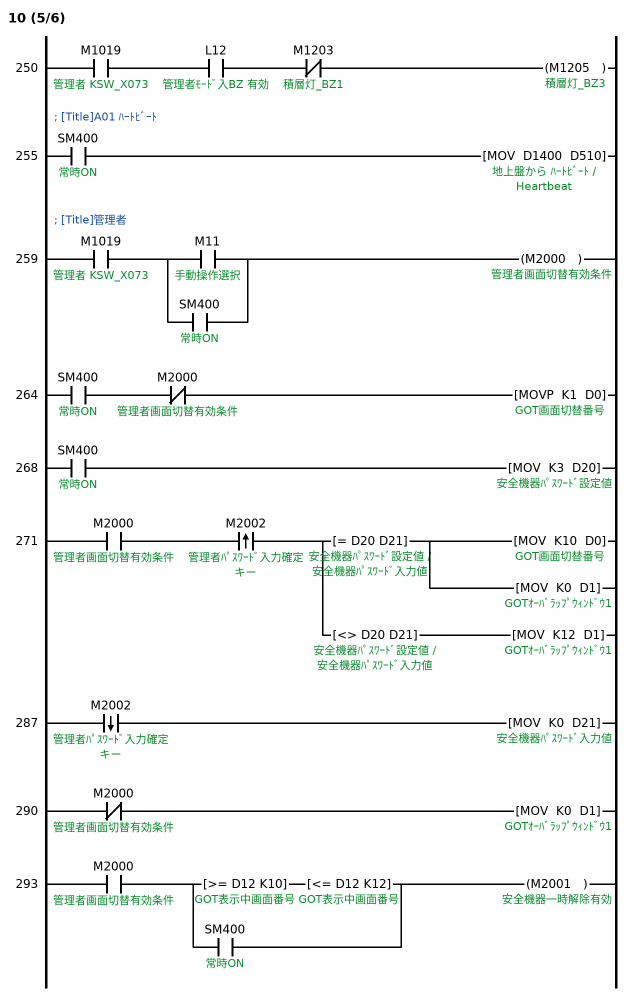
250   LD      M1019  ; 管理者 KSW_X073
      AND     L12  ; 管理者ﾓｰﾄﾞ入BZ 有効
      ANI     M1203  ; 積層灯_BZ1
      OUT     M1205  ; 積層灯_BZ3
; [Title]A01 ﾊｰﾄﾋﾞｰﾄ
255   LD      SM400  ; 常時ON
      MOV     D1400 D510  ; 地上盤から ﾊｰﾄﾋﾞｰﾄ / Heartbeat
; [Title]管理者
259   LD      M1019  ; 管理者 KSW_X073
      LD      M11  ; 手動操作選択
      OR      SM400  ; 常時ON
      ANB
      OUT     M2000  ; 管理者画面切替有効条件
264   LD      SM400  ; 常時ON
      ANI     M2000  ; 管理者画面切替有効条件
      MOVP    K1 D0  ; GOT画面切替番号
268   LD      SM400  ; 常時ON
      MOV     K3 D20  ; 安全機器ﾊﾟｽﾜｰﾄﾞ設定値
271   LD      M2000  ; 管理者画面切替有効条件
      ANDP    M2002  ; 管理者ﾊﾟｽﾜｰﾄﾞ入力確定キー
      MPS
      AND=    D20 D21  ; 安全機器ﾊﾟｽﾜｰﾄﾞ設定値 / 安全機器ﾊﾟｽﾜｰﾄﾞ入力値
      MOV     K10 D0
      MOV     K0 D1  ; GOTｵｰﾊﾞﾗｯﾌﾟｳｨﾝﾄﾞｳ1
      MPP
      AND<>   D20 D21  ; 安全機器ﾊﾟｽﾜｰﾄﾞ設定値 / 安全機器ﾊﾟｽﾜｰﾄﾞ入力値
      MOV     K12 D1
287   LDF     M2002  ; 管理者ﾊﾟｽﾜｰﾄﾞ入力確定キー
      MOV     K0 D21
290   LDI     M2000  ; 管理者画面切替有効条件
      MOV     K0 D1
293   LD      M2000  ; 管理者画面切替有効条件
      LD>=    D12 K10  ; GOT表示中画面番号
      AND<=   D12 K12  ; GOT表示中画面番号
      OR      SM400  ; 常時ON
      ANB
      OUT     M2001  ; 安全機器一時解除有効
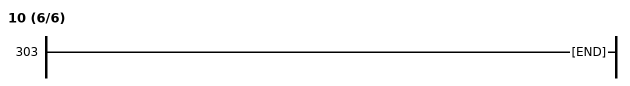
303   END
END_PROGRAM

PROGRAM 11  // 自動搬入
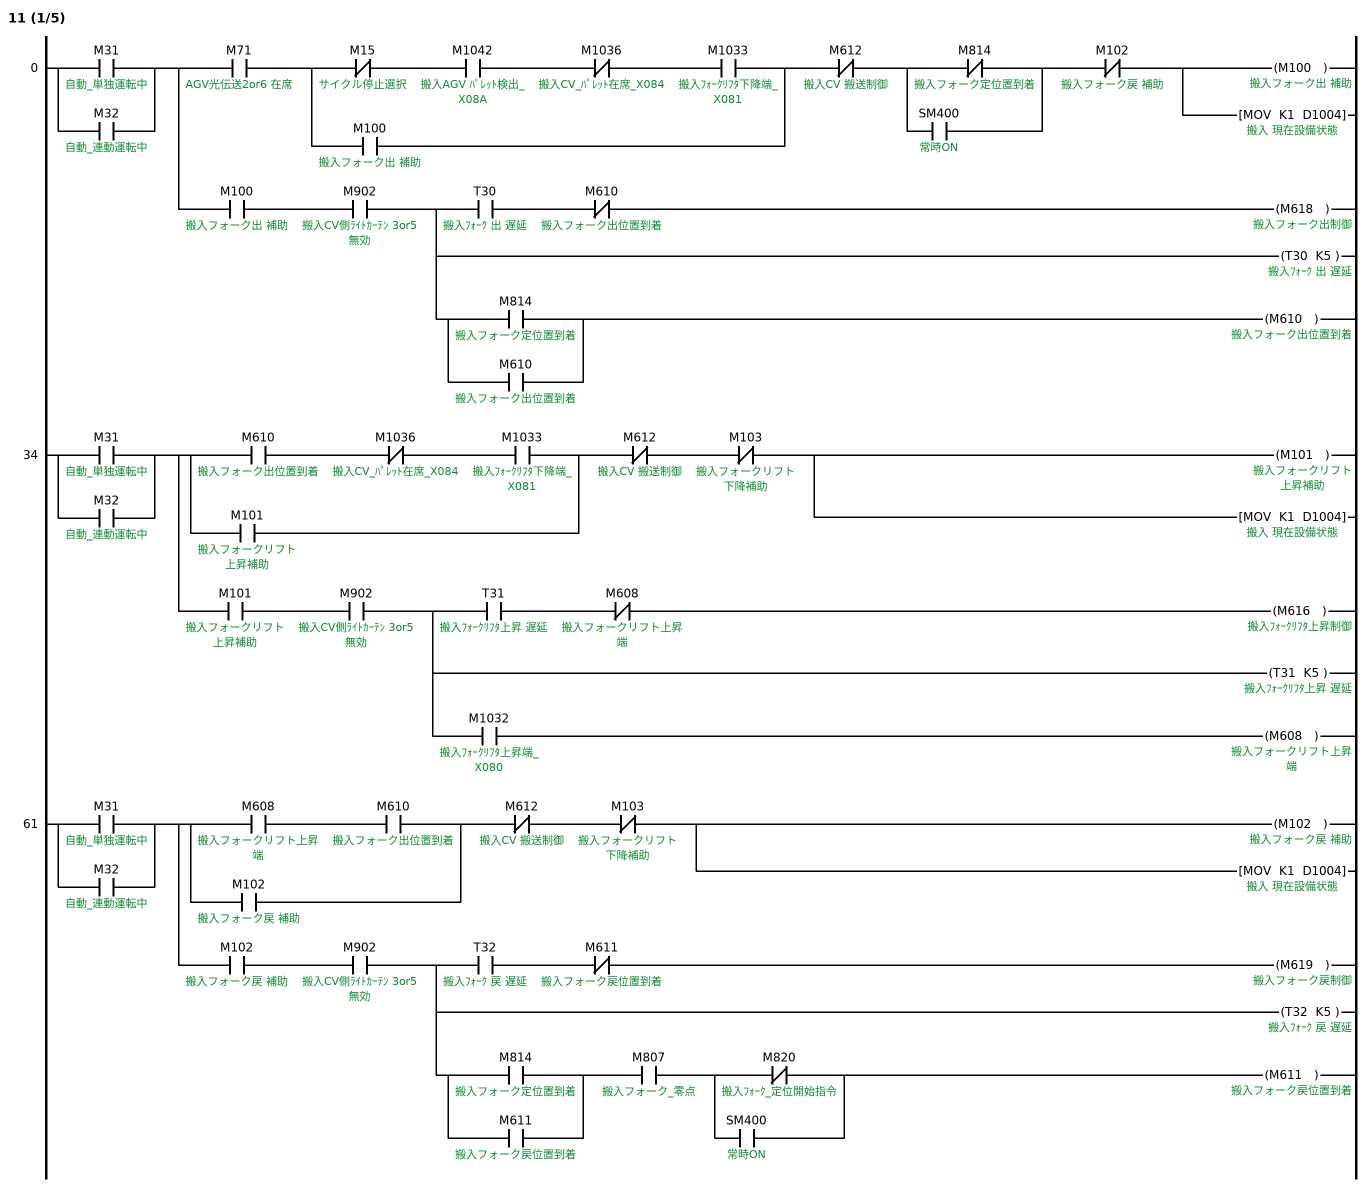
0     LD      M31  ; 自動_単独運転中
      OR      M32  ; 自動_連動運転中
      MPS
      AND     M71  ; AGV光伝送2or6 在席
      LDI     M15  ; サイクル停止選択
      AND     M1042  ; 搬入AGV ﾊﾟﾚｯﾄ検出_X08A
      ANI     M1036  ; 搬入CV_ﾊﾟﾚｯﾄ在席_X084
      AND     M1033  ; 搬入ﾌｫｰｸﾘﾌﾀ下降端_X081
      OR      M100  ; 搬入フォーク出 補助
      ANB
      ANI     M612  ; 搬入CV 搬送制御
      LDI     M814  ; 搬入フォーク定位置到着
      OR      SM400  ; 常時ON
      ANB
      ANI     M102  ; 搬入フォーク戻 補助
      OUT     M100  ; 搬入フォーク出 補助
      MOV     K1 D1004  ; 搬入 現在設備状態
      MPP
      AND     M100  ; 搬入フォーク出 補助
      AND     M902  ; 搬入CV側ﾗｲﾄｶｰﾃﾝ 3or5 無効
      MPS
      AND     T30  ; 搬入ﾌｫｰｸ 出 遅延
      ANI     M610  ; 搬入フォーク出位置到着
      OUT     M618  ; 搬入フォーク出制御
      MPP
      OUT     T30 K5  ; 搬入ﾌｫｰｸ 出 遅延
      LD      M814  ; 搬入フォーク定位置到着
      OR      M610  ; 搬入フォーク出位置到着
      ANB
      OUT     M610  ; 搬入フォーク出位置到着
34    LD      M31  ; 自動_単独運転中
      OR      M32  ; 自動_連動運転中
      MPS
      LD      M610  ; 搬入フォーク出位置到着
      ANI     M1036  ; 搬入CV_ﾊﾟﾚｯﾄ在席_X084
      AND     M1033  ; 搬入ﾌｫｰｸﾘﾌﾀ下降端_X081
      OR      M101  ; 搬入フォークリフト 上昇補助
      ANB
      ANI     M612  ; 搬入CV 搬送制御
      ANI     M103  ; 搬入フォークリフト 下降補助
      OUT     M101  ; 搬入フォークリフト 上昇補助
      MOV     K1 D1004
      MPP
      AND     M101  ; 搬入フォークリフト 上昇補助
      AND     M902  ; 搬入CV側ﾗｲﾄｶｰﾃﾝ 3or5 無効
      MPS
      AND     T31  ; 搬入ﾌｫｰｸﾘﾌﾀ上昇 遅延
      ANI     M608  ; 搬入フォークリフト上昇端
      OUT     M616  ; 搬入ﾌｫｰｸﾘﾌﾀ上昇制御
      MPP
      OUT     T31 K5  ; 搬入ﾌｫｰｸﾘﾌﾀ上昇 遅延
      AND     M1032  ; 搬入ﾌｫｰｸﾘﾌﾀ上昇端_X080
      OUT     M608  ; 搬入フォークリフト上昇端
61    LD      M31  ; 自動_単独運転中
      OR      M32  ; 自動_連動運転中
      MPS
      LD      M608  ; 搬入フォークリフト上昇端
      AND     M610  ; 搬入フォーク出位置到着
      OR      M102  ; 搬入フォーク戻 補助
      ANB
      ANI     M612  ; 搬入CV 搬送制御
      ANI     M103  ; 搬入フォークリフト 下降補助
      OUT     M102  ; 搬入フォーク戻 補助
      MOV     K1 D1004
      MPP
      AND     M102  ; 搬入フォーク戻 補助
      AND     M902  ; 搬入CV側ﾗｲﾄｶｰﾃﾝ 3or5 無効
      MPS
      AND     T32  ; 搬入ﾌｫｰｸ 戻 遅延
      ANI     M611  ; 搬入フォーク戻位置到着
      OUT     M619  ; 搬入フォーク戻制御
      MPP
      OUT     T32 K5  ; 搬入ﾌｫｰｸ 戻 遅延
      LD      M814  ; 搬入フォーク定位置到着
      OR      M611  ; 搬入フォーク戻位置到着
      ANB
      AND     M807  ; 搬入フォーク_零点
      LDI     M820  ; 搬入ﾌｫｰｸ_定位開始指令
      OR      SM400  ; 常時ON
      ANB
      OUT     M611  ; 搬入フォーク戻位置到着
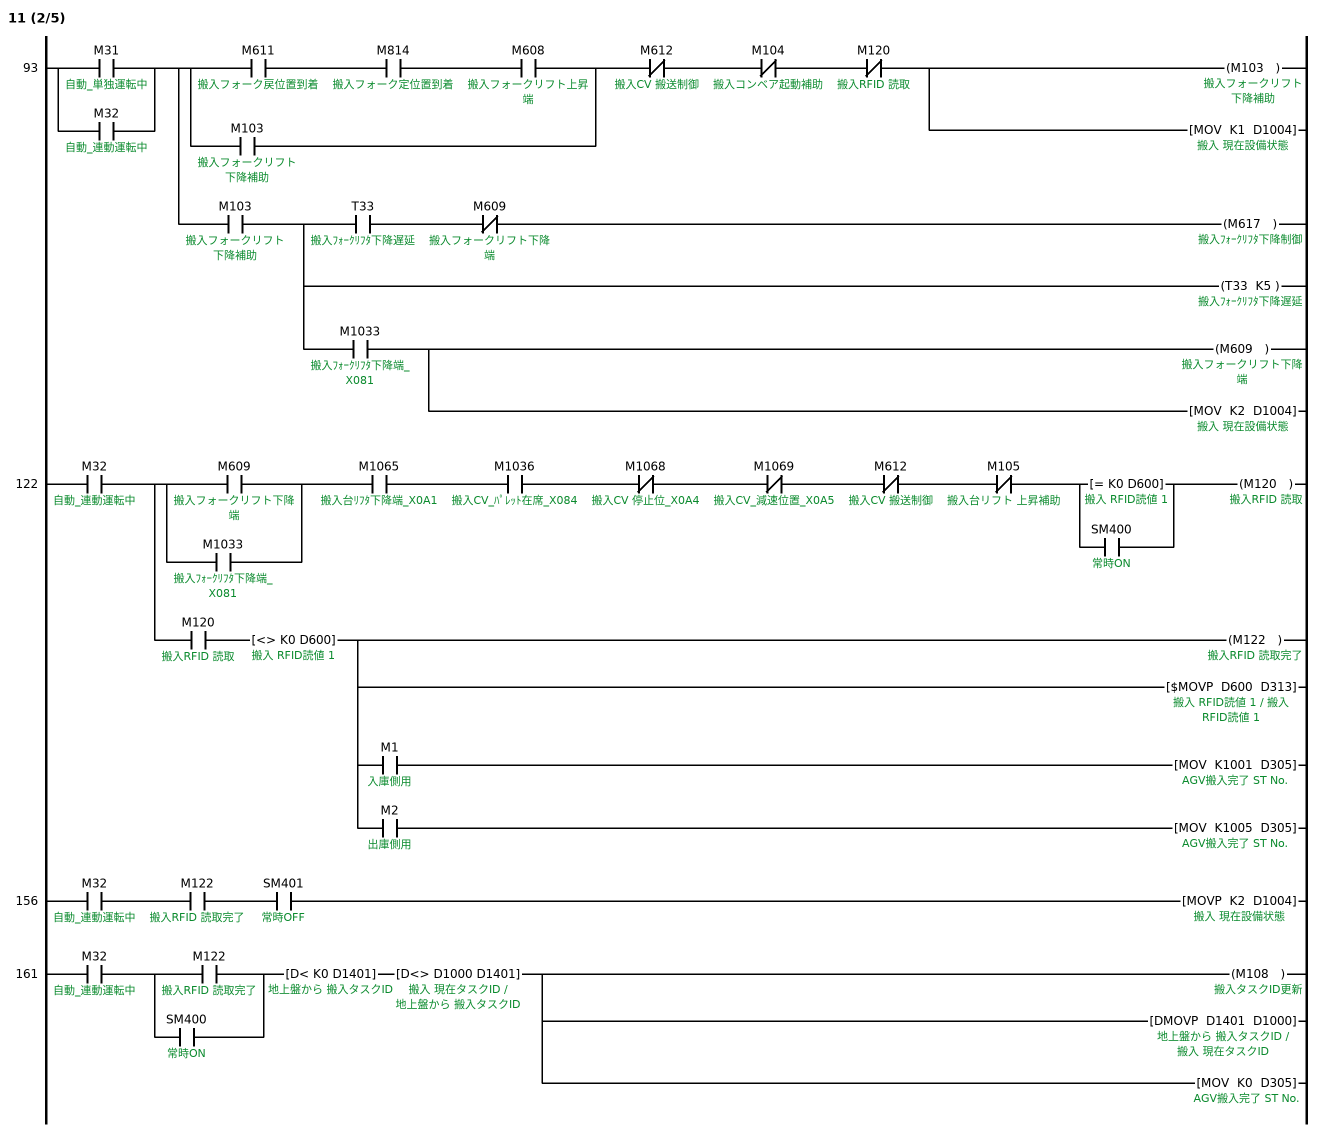
93    LD      M31  ; 自動_単独運転中
      OR      M32  ; 自動_連動運転中
      MPS
      LD      M611  ; 搬入フォーク戻位置到着
      AND     M814  ; 搬入フォーク定位置到着
      AND     M608  ; 搬入フォークリフト上昇端
      OR      M103  ; 搬入フォークリフト 下降補助
      ANB
      ANI     M612  ; 搬入CV 搬送制御
      ANI     M104  ; 搬入コンベア起動補助
      ANI     M120  ; 搬入RFID 読取
      OUT     M103  ; 搬入フォークリフト 下降補助
      MOV     K1 D1004
      MPP
      AND     M103  ; 搬入フォークリフト 下降補助
      MPS
      AND     T33  ; 搬入ﾌｫｰｸﾘﾌﾀ下降遅延
      ANI     M609  ; 搬入フォークリフト下降端
      OUT     M617  ; 搬入ﾌｫｰｸﾘﾌﾀ下降制御
      MPP
      OUT     T33 K5  ; 搬入ﾌｫｰｸﾘﾌﾀ下降遅延
      AND     M1033  ; 搬入ﾌｫｰｸﾘﾌﾀ下降端_X081
      OUT     M609  ; 搬入フォークリフト下降端
      MOV     K2 D1004
122   LD      M32  ; 自動_連動運転中
      MPS
      LD      M609  ; 搬入フォークリフト下降端
      OR      M1033  ; 搬入ﾌｫｰｸﾘﾌﾀ下降端_X081
      ANB
      AND     M1065  ; 搬入台ﾘﾌﾀ下降端_X0A1
      AND     M1036  ; 搬入CV_ﾊﾟﾚｯﾄ在席_X084
      ANI     M1068  ; 搬入CV 停止位_X0A4
      ANI     M1069  ; 搬入CV_減速位置_X0A5
      ANI     M612  ; 搬入CV 搬送制御
      ANI     M105  ; 搬入台リフト 上昇補助
      LD=     K0 D600  ; 搬入 RFID読値 1
      OR      SM400  ; 常時ON
      ANB
      OUT     M120  ; 搬入RFID 読取
      MPP
      AND     M120  ; 搬入RFID 読取
      AND<>   K0 D600  ; 搬入 RFID読値 1
      OUT     M122  ; 搬入RFID 読取完了
      $MOVP   D600 D313  ; 搬入 RFID読値 1
      MPS
      AND     M1  ; 入庫側用
      MOV     K1001 D305  ; AGV搬入完了 ST No.
      MPP
      AND     M2  ; 出庫側用
      MOV     K1005 D305
156   LD      M32  ; 自動_連動運転中
      AND     M122  ; 搬入RFID 読取完了
      AND     SM401  ; 常時OFF
      MOVP    K2 D1004
161   LD      M32  ; 自動_連動運転中
      LD      M122  ; 搬入RFID 読取完了
      OR      SM400  ; 常時ON
      ANB
      ANDD<   K0 D1401  ; 地上盤から 搬入タスクID
      ANDD<>  D1000 D1401  ; 搬入 現在タスクID / 地上盤から 搬入タスクID
      OUT     M108  ; 搬入タスクID更新
      DMOVP   D1401 D1000
      MOV     K0 D305
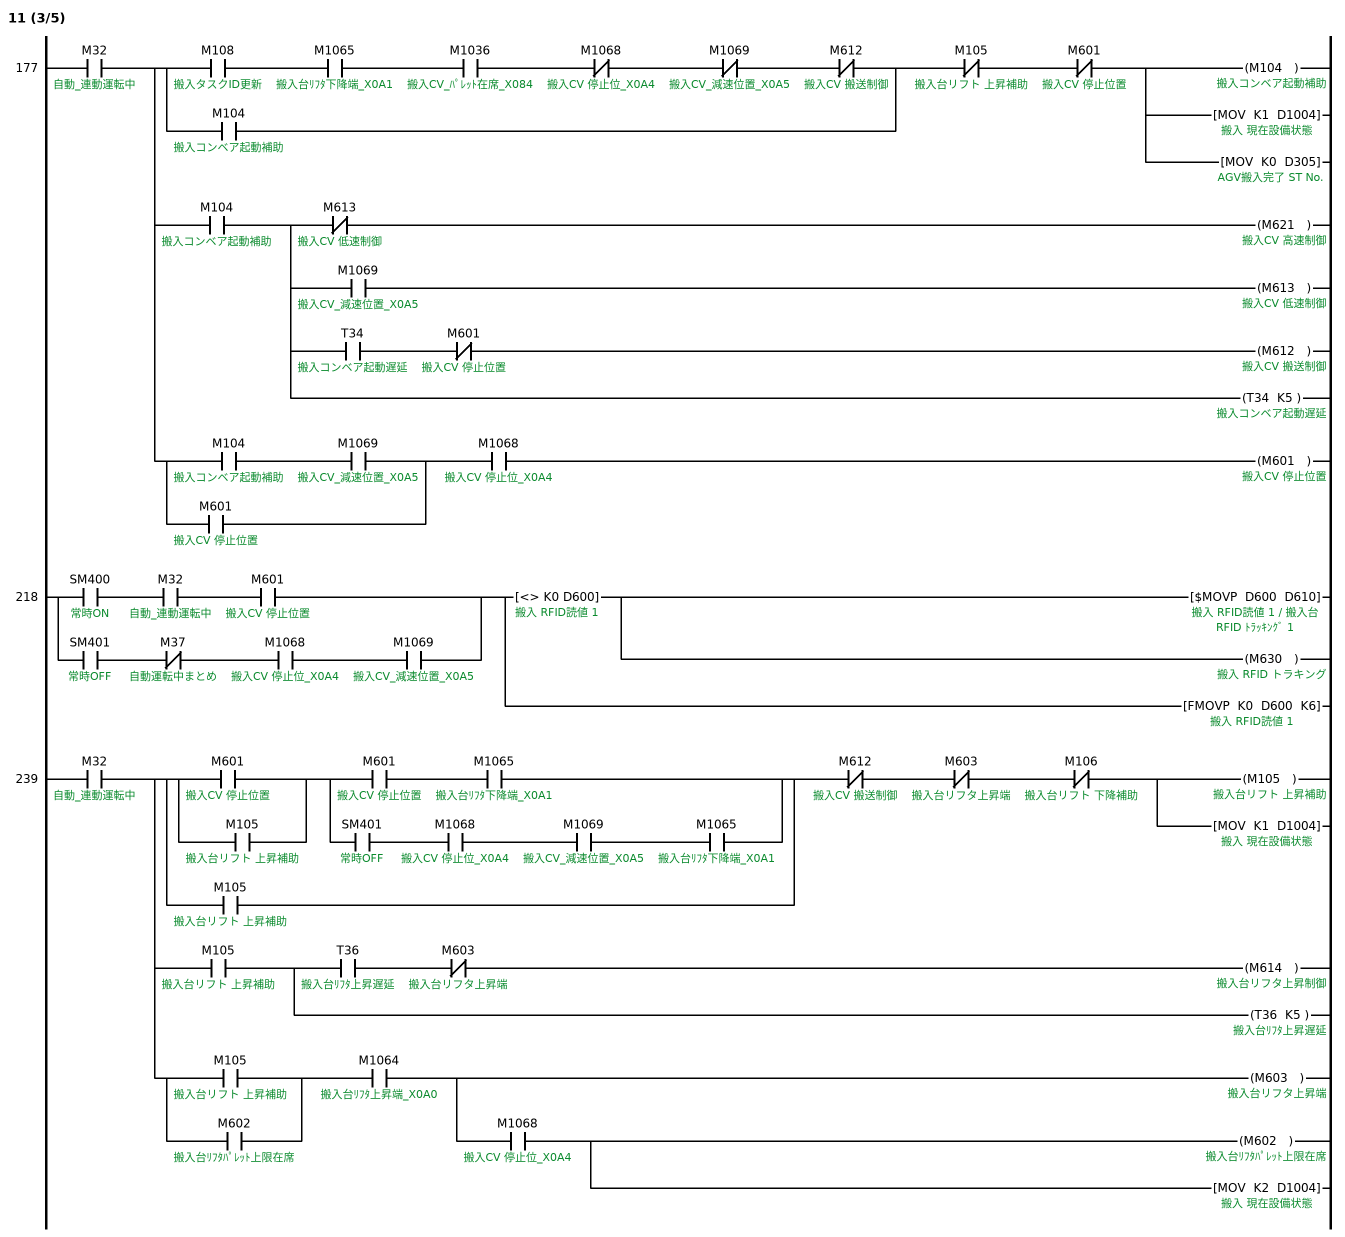
177   LD      M32  ; 自動_連動運転中
      MPS
      LD      M108  ; 搬入タスクID更新
      AND     M1065  ; 搬入台ﾘﾌﾀ下降端_X0A1
      AND     M1036  ; 搬入CV_ﾊﾟﾚｯﾄ在席_X084
      ANI     M1068  ; 搬入CV 停止位_X0A4
      ANI     M1069  ; 搬入CV_減速位置_X0A5
      ANI     M612  ; 搬入CV 搬送制御
      OR      M104  ; 搬入コンベア起動補助
      ANB
      ANI     M105  ; 搬入台リフト 上昇補助
      ANI     M601  ; 搬入CV 停止位置
      OUT     M104  ; 搬入コンベア起動補助
      MOV     K1 D1004
      MOV     K0 D305
      MRD
      AND     M104  ; 搬入コンベア起動補助
      MPS
      ANI     M613  ; 搬入CV 低速制御
      OUT     M621  ; 搬入CV 高速制御
      MRD
      AND     M1069  ; 搬入CV_減速位置_X0A5
      OUT     M613  ; 搬入CV 低速制御
      MRD
      AND     T34  ; 搬入コンベア起動遅延
      ANI     M601  ; 搬入CV 停止位置
      OUT     M612  ; 搬入CV 搬送制御
      MPP
      OUT     T34 K5  ; 搬入コンベア起動遅延
      MPP
      LD      M104  ; 搬入コンベア起動補助
      AND     M1069  ; 搬入CV_減速位置_X0A5
      OR      M601  ; 搬入CV 停止位置
      ANB
      AND     M1068  ; 搬入CV 停止位_X0A4
      OUT     M601  ; 搬入CV 停止位置
218   LD      SM400  ; 常時ON
      AND     M32  ; 自動_連動運転中
      AND     M601  ; 搬入CV 停止位置
      LD      SM401  ; 常時OFF
      ANI     M37  ; 自動運転中まとめ
      AND     M1068  ; 搬入CV 停止位_X0A4
      AND     M1069  ; 搬入CV_減速位置_X0A5
      ORB
      MPS
      AND<>   K0 D600  ; 搬入 RFID読値 1
      $MOVP   D600 D610  ; 搬入台 RFID ﾄﾗｯｷﾝｸﾞ 1
      OUT     M630  ; 搬入 RFID トラキング
      MPP
      FMOVP   K0 D600 K6
239   LD      M32  ; 自動_連動運転中
      MPS
      LD      M601  ; 搬入CV 停止位置
      OR      M105  ; 搬入台リフト 上昇補助
      LD      M601  ; 搬入CV 停止位置
      AND     M1065  ; 搬入台ﾘﾌﾀ下降端_X0A1
      LD      SM401  ; 常時OFF
      AND     M1068  ; 搬入CV 停止位_X0A4
      AND     M1069  ; 搬入CV_減速位置_X0A5
      AND     M1065  ; 搬入台ﾘﾌﾀ下降端_X0A1
      ORB
      ANB
      OR      M105  ; 搬入台リフト 上昇補助
      ANB
      ANI     M612  ; 搬入CV 搬送制御
      ANI     M603  ; 搬入台リフタ上昇端
      ANI     M106  ; 搬入台リフト 下降補助
      OUT     M105  ; 搬入台リフト 上昇補助
      MOV     K1 D1004
      MRD
      AND     M105  ; 搬入台リフト 上昇補助
      MPS
      AND     T36  ; 搬入台ﾘﾌﾀ上昇遅延
      ANI     M603  ; 搬入台リフタ上昇端
      OUT     M614  ; 搬入台リフタ上昇制御
      MPP
      OUT     T36 K5  ; 搬入台ﾘﾌﾀ上昇遅延
      MPP
      LD      M105  ; 搬入台リフト 上昇補助
      OR      M602  ; 搬入台ﾘﾌﾀﾊﾟﾚｯﾄ上限在席
      ANB
      AND     M1064  ; 搬入台ﾘﾌﾀ上昇端_X0A0
      OUT     M603  ; 搬入台リフタ上昇端
      AND     M1068  ; 搬入CV 停止位_X0A4
      OUT     M602  ; 搬入台ﾘﾌﾀﾊﾟﾚｯﾄ上限在席
      MOV     K2 D1004
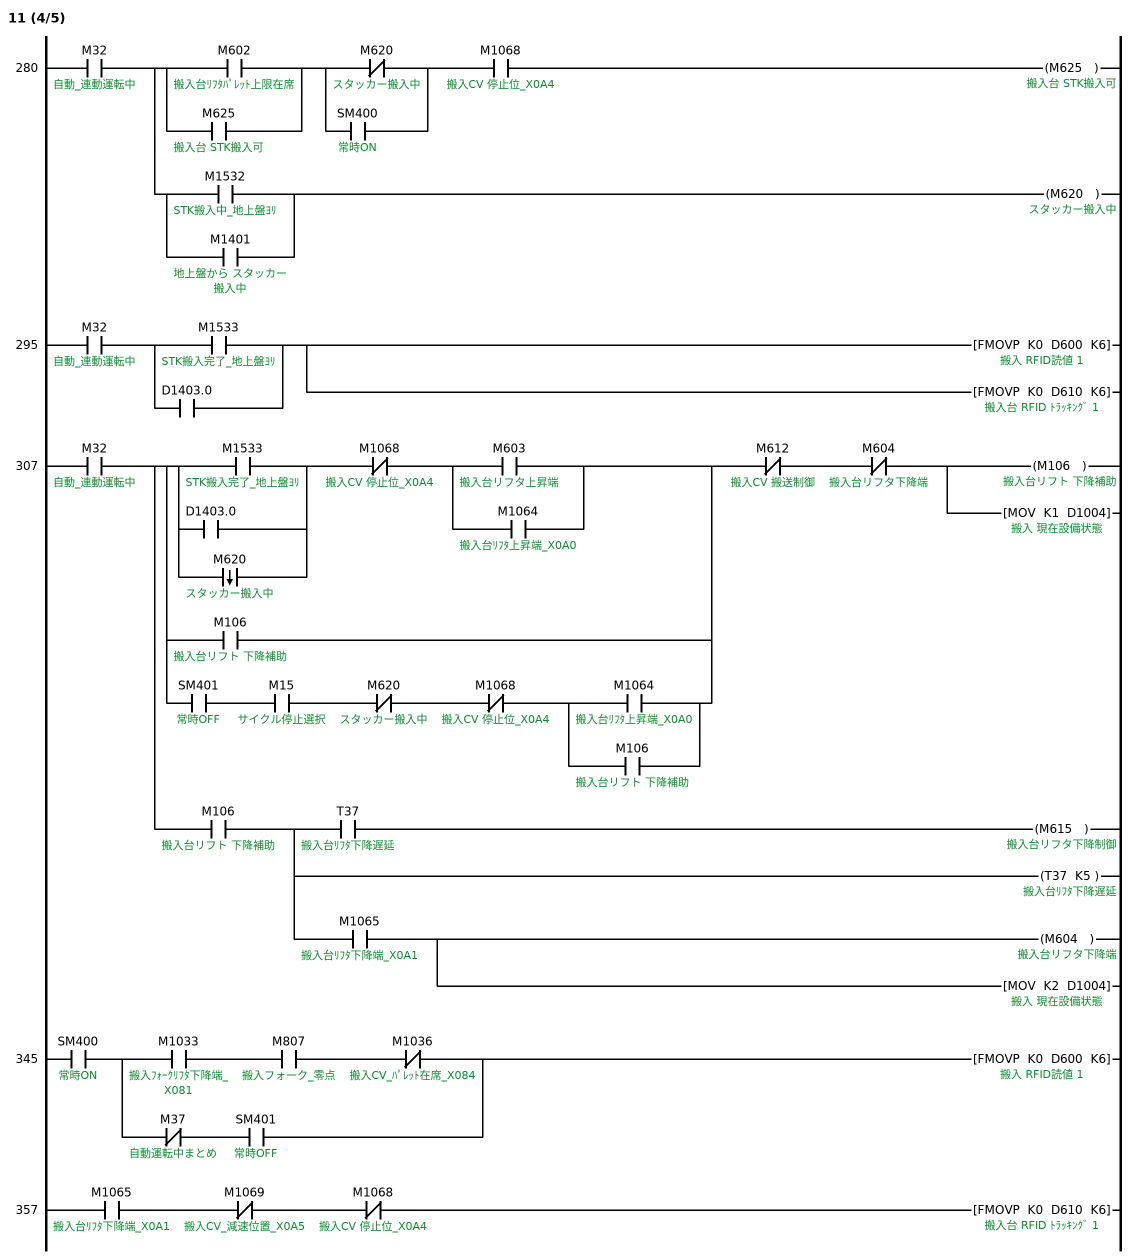
280   LD      M32  ; 自動_連動運転中
      MPS
      LD      M602  ; 搬入台ﾘﾌﾀﾊﾟﾚｯﾄ上限在席
      OR      M625  ; 搬入台 STK搬入可
      ANB
      LDI     M620  ; スタッカー搬入中
      OR      SM400  ; 常時ON
      ANB
      AND     M1068  ; 搬入CV 停止位_X0A4
      OUT     M625  ; 搬入台 STK搬入可
      MPP
      LD      M1532  ; STK搬入中_地上盤ﾖﾘ
      OR      M1401  ; 地上盤から スタッカー 搬入中
      ANB
      OUT     M620  ; スタッカー搬入中
295   LD      M32  ; 自動_連動運転中
      LD      M1533  ; STK搬入完了_地上盤ﾖﾘ
      OR      D1403.0
      ANB
      FMOVP   K0 D600 K6
      FMOVP   K0 D610 K6
307   LD      M32  ; 自動_連動運転中
      MPS
      LD      M1533  ; STK搬入完了_地上盤ﾖﾘ
      OR      D1403.0
      ORF     M620  ; スタッカー搬入中
      ANI     M1068  ; 搬入CV 停止位_X0A4
      LD      M603  ; 搬入台リフタ上昇端
      OR      M1064  ; 搬入台ﾘﾌﾀ上昇端_X0A0
      ANB
      OR      M106  ; 搬入台リフト 下降補助
      LD      SM401  ; 常時OFF
      AND     M15  ; サイクル停止選択
      ANI     M620  ; スタッカー搬入中
      ANI     M1068  ; 搬入CV 停止位_X0A4
      LD      M1064  ; 搬入台ﾘﾌﾀ上昇端_X0A0
      OR      M106  ; 搬入台リフト 下降補助
      ANB
      ORB
      ANB
      ANI     M612  ; 搬入CV 搬送制御
      ANI     M604  ; 搬入台リフタ下降端
      OUT     M106  ; 搬入台リフト 下降補助
      MOV     K1 D1004
      MPP
      AND     M106  ; 搬入台リフト 下降補助
      MPS
      AND     T37  ; 搬入台ﾘﾌﾀ下降遅延
      OUT     M615  ; 搬入台リフタ下降制御
      MPP
      OUT     T37 K5  ; 搬入台ﾘﾌﾀ下降遅延
      AND     M1065  ; 搬入台ﾘﾌﾀ下降端_X0A1
      OUT     M604  ; 搬入台リフタ下降端
      MOV     K2 D1004
345   LD      SM400  ; 常時ON
      LD      M1033  ; 搬入ﾌｫｰｸﾘﾌﾀ下降端_X081
      AND     M807  ; 搬入フォーク_零点
      ANI     M1036  ; 搬入CV_ﾊﾟﾚｯﾄ在席_X084
      LDI     M37  ; 自動運転中まとめ
      AND     SM401  ; 常時OFF
      ORB
      ANB
      FMOVP   K0 D600 K6
357   LD      M1065  ; 搬入台ﾘﾌﾀ下降端_X0A1
      ANI     M1069  ; 搬入CV_減速位置_X0A5
      ANI     M1068  ; 搬入CV 停止位_X0A4
      FMOVP   K0 D610 K6
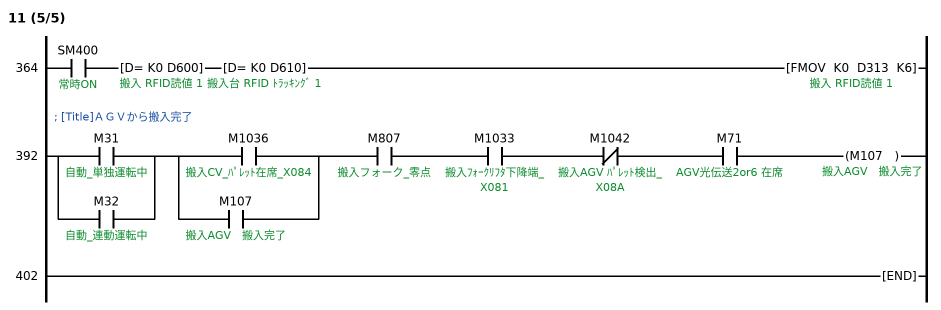
364   LD      SM400  ; 常時ON
      ANDD=   K0 D600  ; 搬入 RFID読値 1
      ANDD=   K0 D610  ; 搬入台 RFID ﾄﾗｯｷﾝｸﾞ 1
      FMOV    K0 D313 K6
; [Title]ＡＧＶから搬入完了
392   LD      M31  ; 自動_単独運転中
      OR      M32  ; 自動_連動運転中
      LD      M1036  ; 搬入CV_ﾊﾟﾚｯﾄ在席_X084
      OR      M107  ; 搬入AGV　搬入完了
      ANB
      AND     M807  ; 搬入フォーク_零点
      AND     M1033  ; 搬入ﾌｫｰｸﾘﾌﾀ下降端_X081
      ANI     M1042  ; 搬入AGV ﾊﾟﾚｯﾄ検出_X08A
      AND     M71  ; AGV光伝送2or6 在席
      OUT     M107  ; 搬入AGV　搬入完了
402   END
END_PROGRAM

PROGRAM 12  // 自動搬出
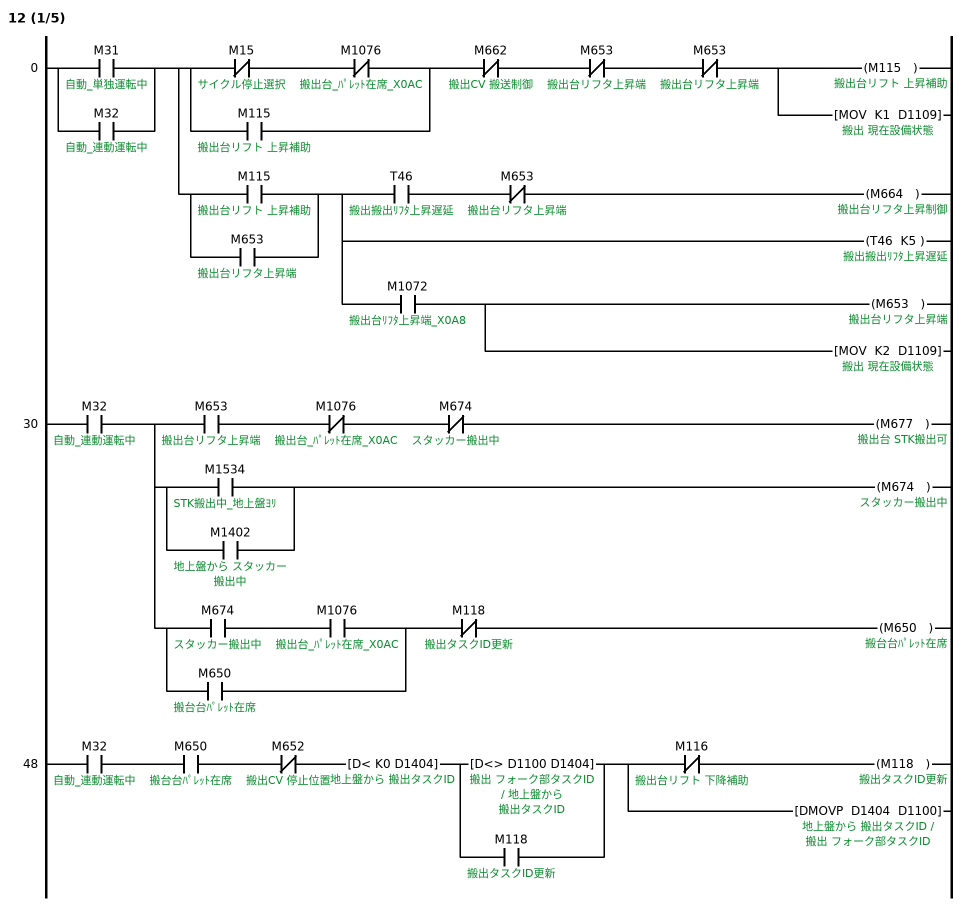
0     LD      M31  ; 自動_単独運転中
      OR      M32  ; 自動_連動運転中
      MPS
      LDI     M15  ; サイクル停止選択
      ANI     M1076  ; 搬出台_ﾊﾟﾚｯﾄ在席_X0AC
      OR      M115  ; 搬出台リフト 上昇補助
      ANB
      ANI     M662  ; 搬出CV 搬送制御
      ANI     M653  ; 搬出台リフタ上昇端
      ANI     M653  ; 搬出台リフタ上昇端
      OUT     M115  ; 搬出台リフト 上昇補助
      MOV     K1 D1109  ; 搬出 現在設備状態
      MPP
      LD      M115  ; 搬出台リフト 上昇補助
      OR      M653  ; 搬出台リフタ上昇端
      ANB
      MPS
      AND     T46  ; 搬出搬出ﾘﾌﾀ上昇遅延
      ANI     M653  ; 搬出台リフタ上昇端
      OUT     M664  ; 搬出台リフタ上昇制御
      MPP
      OUT     T46 K5  ; 搬出搬出ﾘﾌﾀ上昇遅延
      AND     M1072  ; 搬出台ﾘﾌﾀ上昇端_X0A8
      OUT     M653  ; 搬出台リフタ上昇端
      MOV     K2 D1109
30    LD      M32  ; 自動_連動運転中
      MPS
      AND     M653  ; 搬出台リフタ上昇端
      ANI     M1076  ; 搬出台_ﾊﾟﾚｯﾄ在席_X0AC
      ANI     M674  ; スタッカー搬出中
      OUT     M677  ; 搬出台 STK搬出可
      MRD
      LD      M1534  ; STK搬出中_地上盤ﾖﾘ
      OR      M1402  ; 地上盤から スタッカー 搬出中
      ANB
      OUT     M674  ; スタッカー搬出中
      MPP
      LD      M674  ; スタッカー搬出中
      AND     M1076  ; 搬出台_ﾊﾟﾚｯﾄ在席_X0AC
      OR      M650  ; 搬台台ﾊﾟﾚｯﾄ在席
      ANB
      ANI     M118  ; 搬出タスクID更新
      OUT     M650  ; 搬台台ﾊﾟﾚｯﾄ在席
48    LD      M32  ; 自動_連動運転中
      AND     M650  ; 搬台台ﾊﾟﾚｯﾄ在席
      ANI     M652  ; 搬出CV 停止位置
      ANDD<   K0 D1404  ; 地上盤から 搬出タスクID
      LDD<>   D1100 D1404  ; 搬出 フォーク部タスクID / 地上盤から 搬出タスクID
      OR      M118  ; 搬出タスクID更新
      ANB
      MPS
      ANI     M116  ; 搬出台リフト 下降補助
      OUT     M118  ; 搬出タスクID更新
      MPP
      DMOVP   D1404 D1100
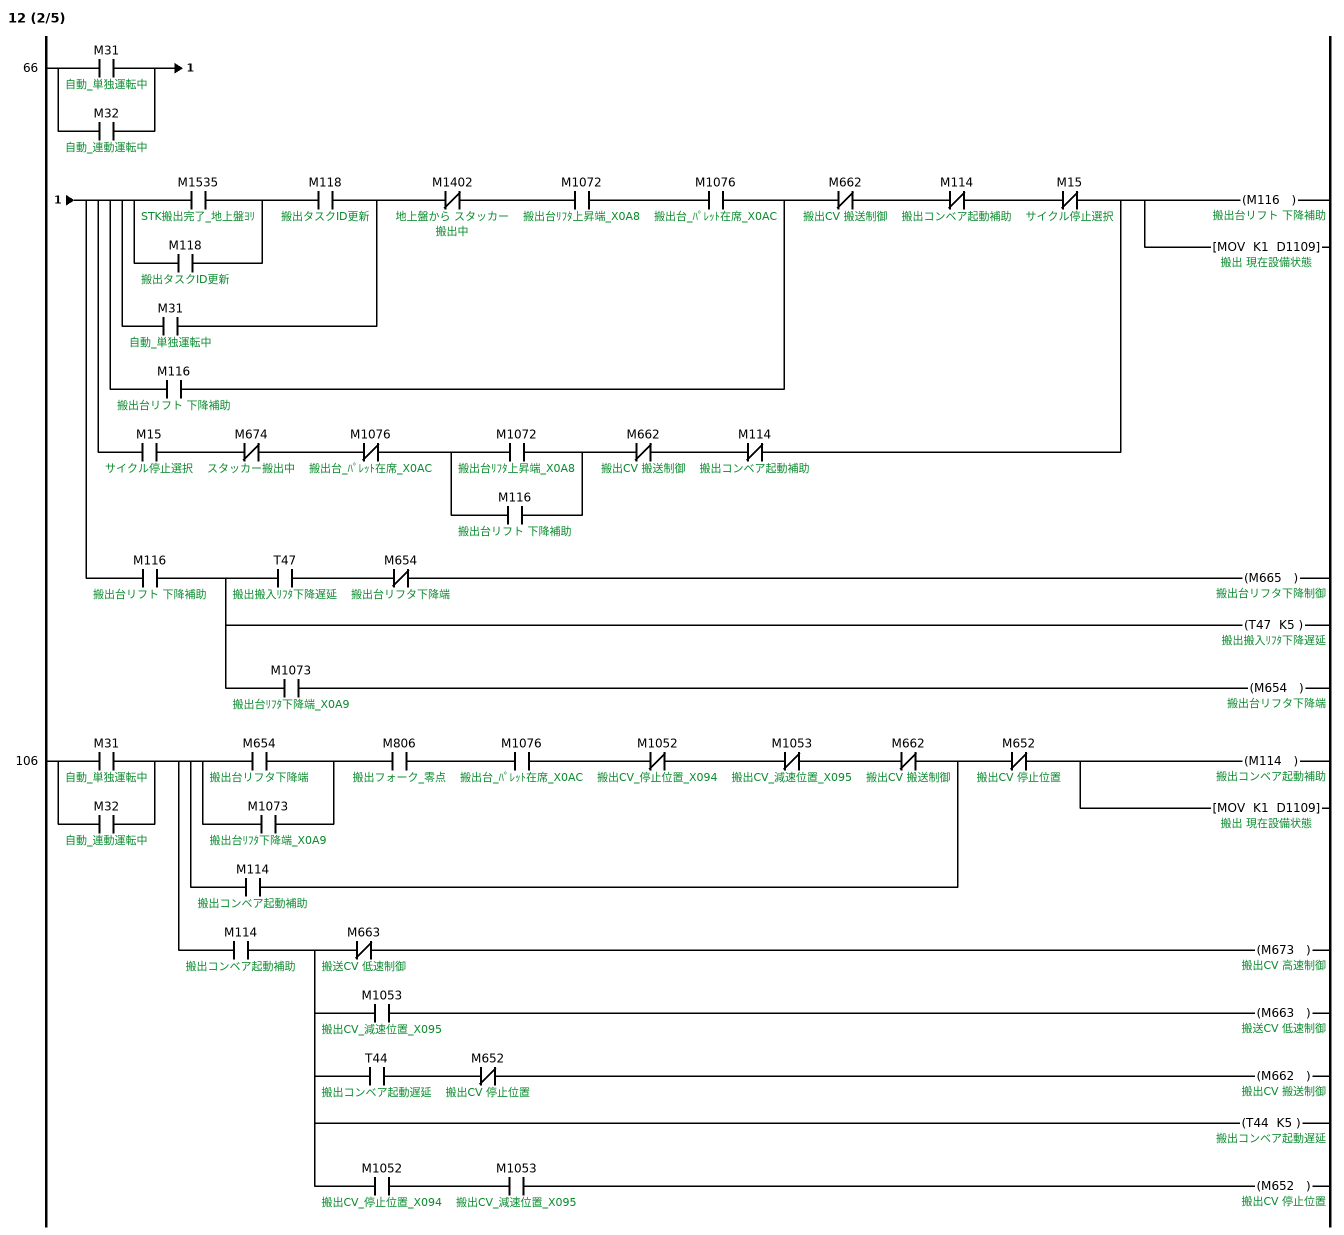
66    LD      M31  ; 自動_単独運転中
      OR      M32  ; 自動_連動運転中
      MPS
      LD      M1535  ; STK搬出完了_地上盤ﾖﾘ
      OR      M118  ; 搬出タスクID更新
      AND     M118  ; 搬出タスクID更新
      OR      M31  ; 自動_単独運転中
      ANI     M1402  ; 地上盤から スタッカー 搬出中
      AND     M1072  ; 搬出台ﾘﾌﾀ上昇端_X0A8
      AND     M1076  ; 搬出台_ﾊﾟﾚｯﾄ在席_X0AC
      OR      M116  ; 搬出台リフト 下降補助
      ANI     M662  ; 搬出CV 搬送制御
      ANI     M114  ; 搬出コンベア起動補助
      ANI     M15  ; サイクル停止選択
      LD      M15  ; サイクル停止選択
      ANI     M674  ; スタッカー搬出中
      ANI     M1076  ; 搬出台_ﾊﾟﾚｯﾄ在席_X0AC
      LD      M1072  ; 搬出台ﾘﾌﾀ上昇端_X0A8
      OR      M116  ; 搬出台リフト 下降補助
      ANB
      ANI     M662  ; 搬出CV 搬送制御
      ANI     M114  ; 搬出コンベア起動補助
      ORB
      ANB
      OUT     M116  ; 搬出台リフト 下降補助
      MOV     K1 D1109
      MPP
      AND     M116  ; 搬出台リフト 下降補助
      MPS
      AND     T47  ; 搬出搬入ﾘﾌﾀ下降遅延
      ANI     M654  ; 搬出台リフタ下降端
      OUT     M665  ; 搬出台リフタ下降制御
      MPP
      OUT     T47 K5  ; 搬出搬入ﾘﾌﾀ下降遅延
      AND     M1073  ; 搬出台ﾘﾌﾀ下降端_X0A9
      OUT     M654  ; 搬出台リフタ下降端
106   LD      M31  ; 自動_単独運転中
      OR      M32  ; 自動_連動運転中
      MPS
      LD      M654  ; 搬出台リフタ下降端
      OR      M1073  ; 搬出台ﾘﾌﾀ下降端_X0A9
      AND     M806  ; 搬出フォーク_零点
      AND     M1076  ; 搬出台_ﾊﾟﾚｯﾄ在席_X0AC
      ANI     M1052  ; 搬出CV_停止位置_X094
      ANI     M1053  ; 搬出CV_減速位置_X095
      ANI     M662  ; 搬出CV 搬送制御
      OR      M114  ; 搬出コンベア起動補助
      ANB
      ANI     M652  ; 搬出CV 停止位置
      OUT     M114  ; 搬出コンベア起動補助
      MOV     K1 D1109
      MPP
      AND     M114  ; 搬出コンベア起動補助
      MPS
      ANI     M663  ; 搬送CV 低速制御
      OUT     M673  ; 搬出CV 高速制御
      MRD
      AND     M1053  ; 搬出CV_減速位置_X095
      OUT     M663  ; 搬送CV 低速制御
      MRD
      AND     T44  ; 搬出コンベア起動遅延
      ANI     M652  ; 搬出CV 停止位置
      OUT     M662  ; 搬出CV 搬送制御
      MPP
      OUT     T44 K5  ; 搬出コンベア起動遅延
      AND     M1052  ; 搬出CV_停止位置_X094
      AND     M1053  ; 搬出CV_減速位置_X095
      OUT     M652  ; 搬出CV 停止位置
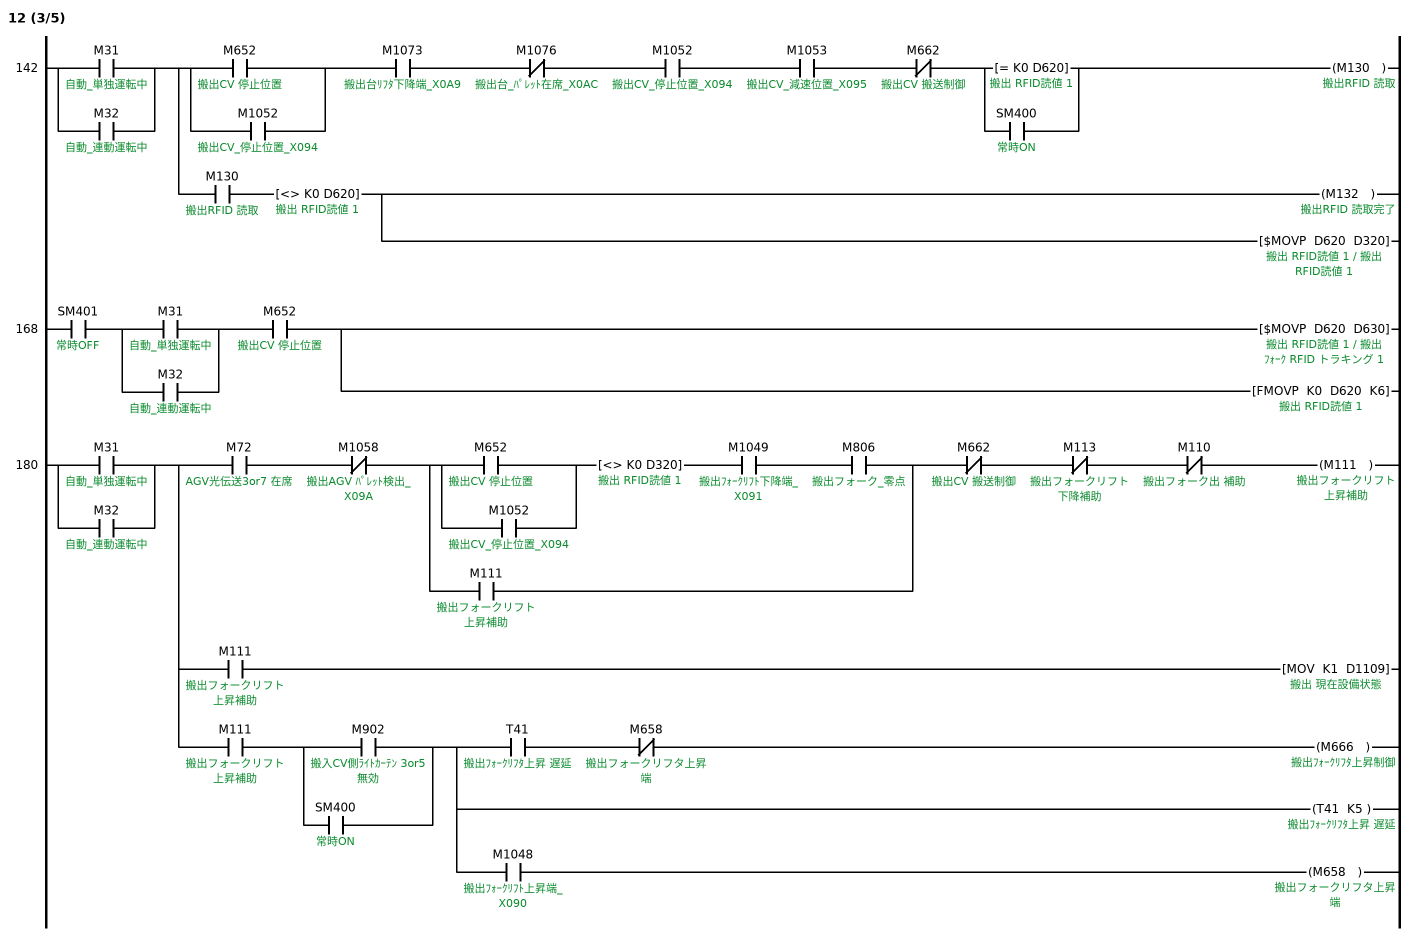
142   LD      M31  ; 自動_単独運転中
      OR      M32  ; 自動_連動運転中
      MPS
      LD      M652  ; 搬出CV 停止位置
      OR      M1052  ; 搬出CV_停止位置_X094
      ANB
      AND     M1073  ; 搬出台ﾘﾌﾀ下降端_X0A9
      ANI     M1076  ; 搬出台_ﾊﾟﾚｯﾄ在席_X0AC
      AND     M1052  ; 搬出CV_停止位置_X094
      AND     M1053  ; 搬出CV_減速位置_X095
      ANI     M662  ; 搬出CV 搬送制御
      LD=     K0 D620  ; 搬出 RFID読値 1
      OR      SM400  ; 常時ON
      ANB
      OUT     M130  ; 搬出RFID 読取
      MPP
      AND     M130  ; 搬出RFID 読取
      AND<>   K0 D620  ; 搬出 RFID読値 1
      OUT     M132  ; 搬出RFID 読取完了
      $MOVP   D620 D320  ; 搬出 RFID読値 1
168   LD      SM401  ; 常時OFF
      LD      M31  ; 自動_単独運転中
      OR      M32  ; 自動_連動運転中
      ANB
      AND     M652  ; 搬出CV 停止位置
      $MOVP   D620 D630  ; 搬出 ﾌｫｰｸ RFID トラキング 1
      FMOVP   K0 D620 K6
180   LD      M31  ; 自動_単独運転中
      OR      M32  ; 自動_連動運転中
      MPS
      AND     M72  ; AGV光伝送3or7 在席
      ANI     M1058  ; 搬出AGV ﾊﾟﾚｯﾄ検出_X09A
      LD      M652  ; 搬出CV 停止位置
      OR      M1052  ; 搬出CV_停止位置_X094
      AND<>   K0 D320  ; 搬出 RFID読値 1
      AND     M1049  ; 搬出ﾌｫｰｸﾘﾌﾄ下降端_X091
      AND     M806  ; 搬出フォーク_零点
      OR      M111  ; 搬出フォークリフト 上昇補助
      ANB
      ANI     M662  ; 搬出CV 搬送制御
      ANI     M113  ; 搬出フォークリフト 下降補助
      ANI     M110  ; 搬出フォーク出 補助
      OUT     M111  ; 搬出フォークリフト 上昇補助
      MRD
      AND     M111  ; 搬出フォークリフト 上昇補助
      MOV     K1 D1109
      MPP
      AND     M111  ; 搬出フォークリフト 上昇補助
      LD      M902  ; 搬入CV側ﾗｲﾄｶｰﾃﾝ 3or5 無効
      OR      SM400  ; 常時ON
      ANB
      MPS
      AND     T41  ; 搬出ﾌｫｰｸﾘﾌﾀ上昇 遅延
      ANI     M658  ; 搬出フォークリフタ上昇端
      OUT     M666  ; 搬出ﾌｫｰｸﾘﾌﾀ上昇制御
      MPP
      OUT     T41 K5  ; 搬出ﾌｫｰｸﾘﾌﾀ上昇 遅延
      AND     M1048  ; 搬出ﾌｫｰｸﾘﾌﾄ上昇端_X090
      OUT     M658  ; 搬出フォークリフタ上昇端
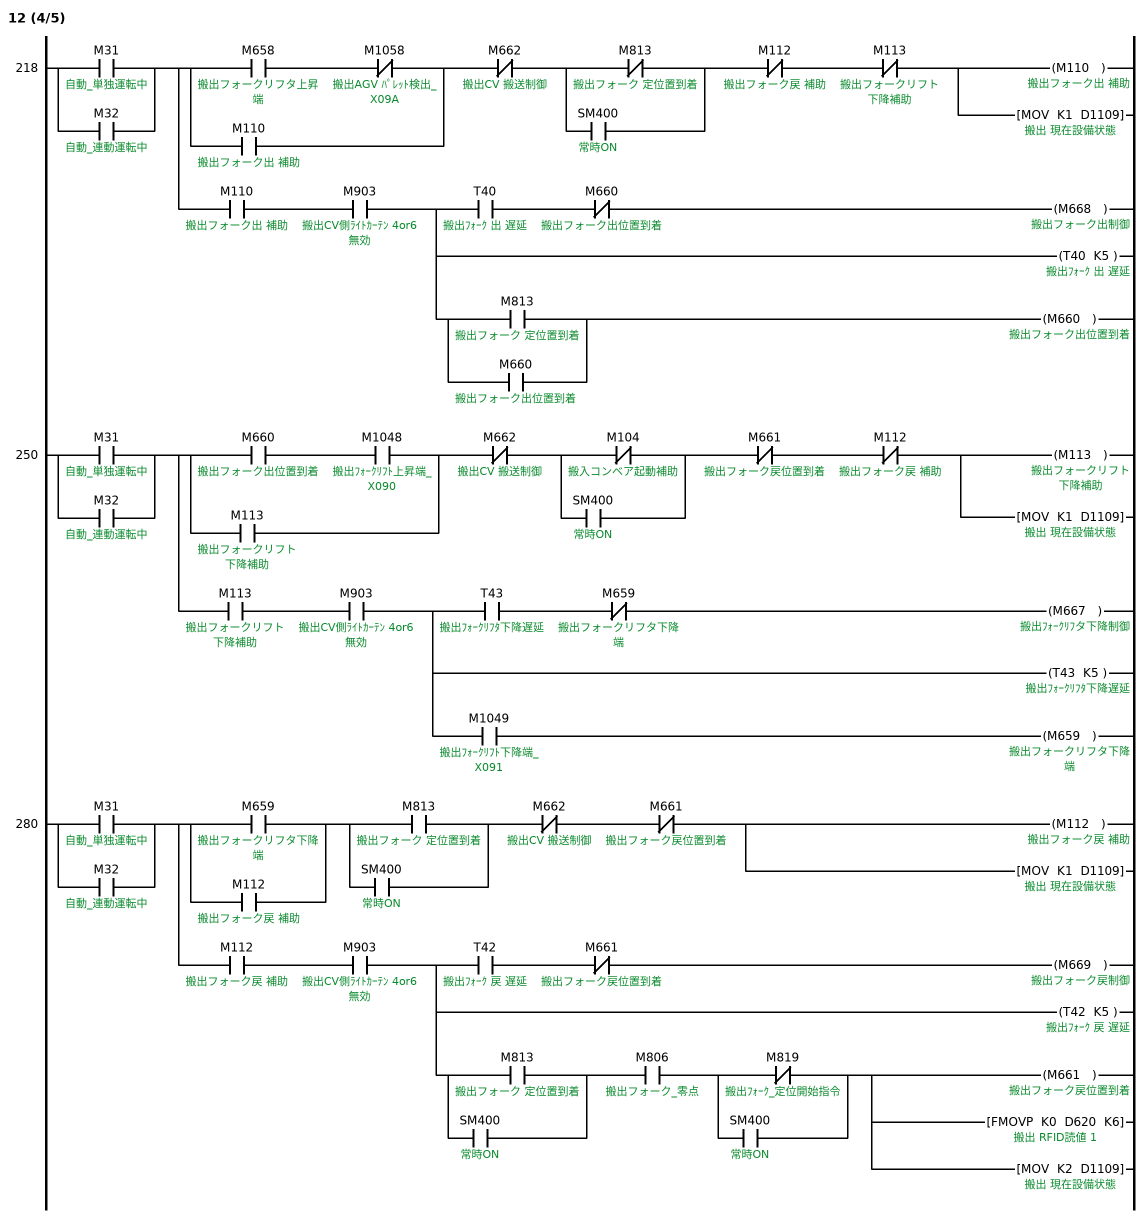
218   LD      M31  ; 自動_単独運転中
      OR      M32  ; 自動_連動運転中
      MPS
      LD      M658  ; 搬出フォークリフタ上昇端
      ANI     M1058  ; 搬出AGV ﾊﾟﾚｯﾄ検出_X09A
      OR      M110  ; 搬出フォーク出 補助
      ANB
      ANI     M662  ; 搬出CV 搬送制御
      LDI     M813  ; 搬出フォーク 定位置到着
      OR      SM400  ; 常時ON
      ANB
      ANI     M112  ; 搬出フォーク戻 補助
      ANI     M113  ; 搬出フォークリフト 下降補助
      OUT     M110  ; 搬出フォーク出 補助
      MOV     K1 D1109
      MPP
      AND     M110  ; 搬出フォーク出 補助
      AND     M903  ; 搬出CV側ﾗｲﾄｶｰﾃﾝ 4or6 無効
      MPS
      AND     T40  ; 搬出ﾌｫｰｸ 出 遅延
      ANI     M660  ; 搬出フォーク出位置到着
      OUT     M668  ; 搬出フォーク出制御
      MPP
      OUT     T40 K5  ; 搬出ﾌｫｰｸ 出 遅延
      LD      M813  ; 搬出フォーク 定位置到着
      OR      M660  ; 搬出フォーク出位置到着
      ANB
      OUT     M660  ; 搬出フォーク出位置到着
250   LD      M31  ; 自動_単独運転中
      OR      M32  ; 自動_連動運転中
      MPS
      LD      M660  ; 搬出フォーク出位置到着
      AND     M1048  ; 搬出ﾌｫｰｸﾘﾌﾄ上昇端_X090
      OR      M113  ; 搬出フォークリフト 下降補助
      ANB
      ANI     M662  ; 搬出CV 搬送制御
      LDI     M104  ; 搬入コンベア起動補助
      OR      SM400  ; 常時ON
      ANB
      ANI     M661  ; 搬出フォーク戻位置到着
      ANI     M112  ; 搬出フォーク戻 補助
      OUT     M113  ; 搬出フォークリフト 下降補助
      MOV     K1 D1109
      MPP
      AND     M113  ; 搬出フォークリフト 下降補助
      AND     M903  ; 搬出CV側ﾗｲﾄｶｰﾃﾝ 4or6 無効
      MPS
      AND     T43  ; 搬出ﾌｫｰｸﾘﾌﾀ下降遅延
      ANI     M659  ; 搬出フォークリフタ下降端
      OUT     M667  ; 搬出ﾌｫｰｸﾘﾌタ下降制御
      MPP
      OUT     T43 K5  ; 搬出ﾌｫｰｸﾘﾌﾀ下降遅延
      AND     M1049  ; 搬出ﾌｫｰｸﾘﾌﾄ下降端_X091
      OUT     M659  ; 搬出フォークリフタ下降端
280   LD      M31  ; 自動_単独運転中
      OR      M32  ; 自動_連動運転中
      MPS
      LD      M659  ; 搬出フォークリフタ下降端
      OR      M112  ; 搬出フォーク戻 補助
      ANB
      LD      M813  ; 搬出フォーク 定位置到着
      OR      SM400  ; 常時ON
      ANB
      ANI     M662  ; 搬出CV 搬送制御
      ANI     M661  ; 搬出フォーク戻位置到着
      OUT     M112  ; 搬出フォーク戻 補助
      MOV     K1 D1109
      MPP
      AND     M112  ; 搬出フォーク戻 補助
      AND     M903  ; 搬出CV側ﾗｲﾄｶｰﾃﾝ 4or6 無効
      MPS
      AND     T42  ; 搬出ﾌｫｰｸ 戻 遅延
      ANI     M661  ; 搬出フォーク戻位置到着
      OUT     M669  ; 搬出フォーク戻制御
      MPP
      OUT     T42 K5  ; 搬出ﾌｫｰｸ 戻 遅延
      LD      M813  ; 搬出フォーク 定位置到着
      OR      SM400  ; 常時ON
      ANB
      AND     M806  ; 搬出フォーク_零点
      LDI     M819  ; 搬出ﾌｫｰｸ_定位開始指令
      OR      SM400  ; 常時ON
      ANB
      OUT     M661  ; 搬出フォーク戻位置到着
      FMOVP   K0 D620 K6
      MOV     K2 D1109
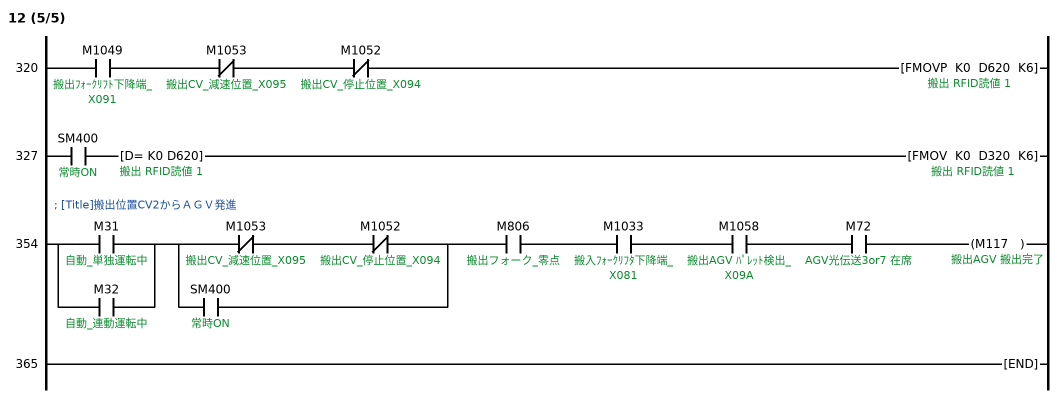
320   LD      M1049  ; 搬出ﾌｫｰｸﾘﾌﾄ下降端_X091
      ANI     M1053  ; 搬出CV_減速位置_X095
      ANI     M1052  ; 搬出CV_停止位置_X094
      FMOVP   K0 D620 K6
327   LD      SM400  ; 常時ON
      ANDD=   K0 D620  ; 搬出 RFID読値 1
      FMOV    K0 D320 K6
; [Title]搬出位置CV2からＡＧＶ発進
354   LD      M31  ; 自動_単独運転中
      OR      M32  ; 自動_連動運転中
      LDI     M1053  ; 搬出CV_減速位置_X095
      ANI     M1052  ; 搬出CV_停止位置_X094
      OR      SM400  ; 常時ON
      ANB
      AND     M806  ; 搬出フォーク_零点
      AND     M1033  ; 搬入ﾌｫｰｸﾘﾌﾀ下降端_X081
      AND     M1058  ; 搬出AGV ﾊﾟﾚｯﾄ検出_X09A
      AND     M72  ; AGV光伝送3or7 在席
      OUT     M117  ; 搬出AGV 搬出完了
365   END
END_PROGRAM

PROGRAM 13  // 手動操作
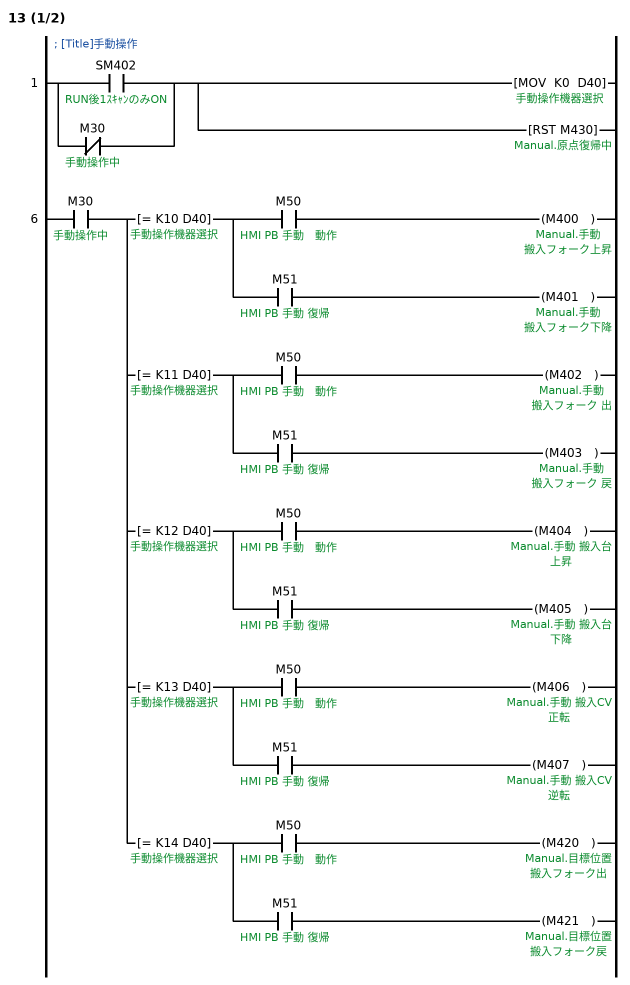
; [Title]手動操作
1     LD      SM402  ; RUN後1ｽｷｬﾝのみON
      ORI     M30  ; 手動操作中
      MOV     K0 D40  ; 手動操作機器選択
      RST     M430  ; Manual.原点復帰中
6     LD      M30  ; 手動操作中
      MPS
      AND=    K10 D40  ; 手動操作機器選択
      MPS
      AND     M50  ; HMI PB 手動　動作
      OUT     M400  ; Manual.手動 搬入フォーク上昇
      MPP
      AND     M51  ; HMI PB 手動 復帰
      OUT     M401  ; Manual.手動 搬入フォーク下降
      MRD
      AND=    K11 D40  ; 手動操作機器選択
      MPS
      AND     M50  ; HMI PB 手動　動作
      OUT     M402  ; Manual.手動 搬入フォーク 出
      MPP
      AND     M51  ; HMI PB 手動 復帰
      OUT     M403  ; Manual.手動 搬入フォーク 戻
      MRD
      AND=    K12 D40  ; 手動操作機器選択
      MPS
      AND     M50  ; HMI PB 手動　動作
      OUT     M404  ; Manual.手動 搬入台 上昇
      MPP
      AND     M51  ; HMI PB 手動 復帰
      OUT     M405  ; Manual.手動 搬入台 下降
      MRD
      AND=    K13 D40  ; 手動操作機器選択
      MPS
      AND     M50  ; HMI PB 手動　動作
      OUT     M406  ; Manual.手動 搬入CV 正転
      MPP
      AND     M51  ; HMI PB 手動 復帰
      OUT     M407  ; Manual.手動 搬入CV 逆転
      MPP
      AND=    K14 D40  ; 手動操作機器選択
      MPS
      AND     M50  ; HMI PB 手動　動作
      OUT     M420  ; Manual.目標位置 搬入フォーク出
      MPP
      AND     M51  ; HMI PB 手動 復帰
      OUT     M421  ; Manual.目標位置 搬入フォーク戻
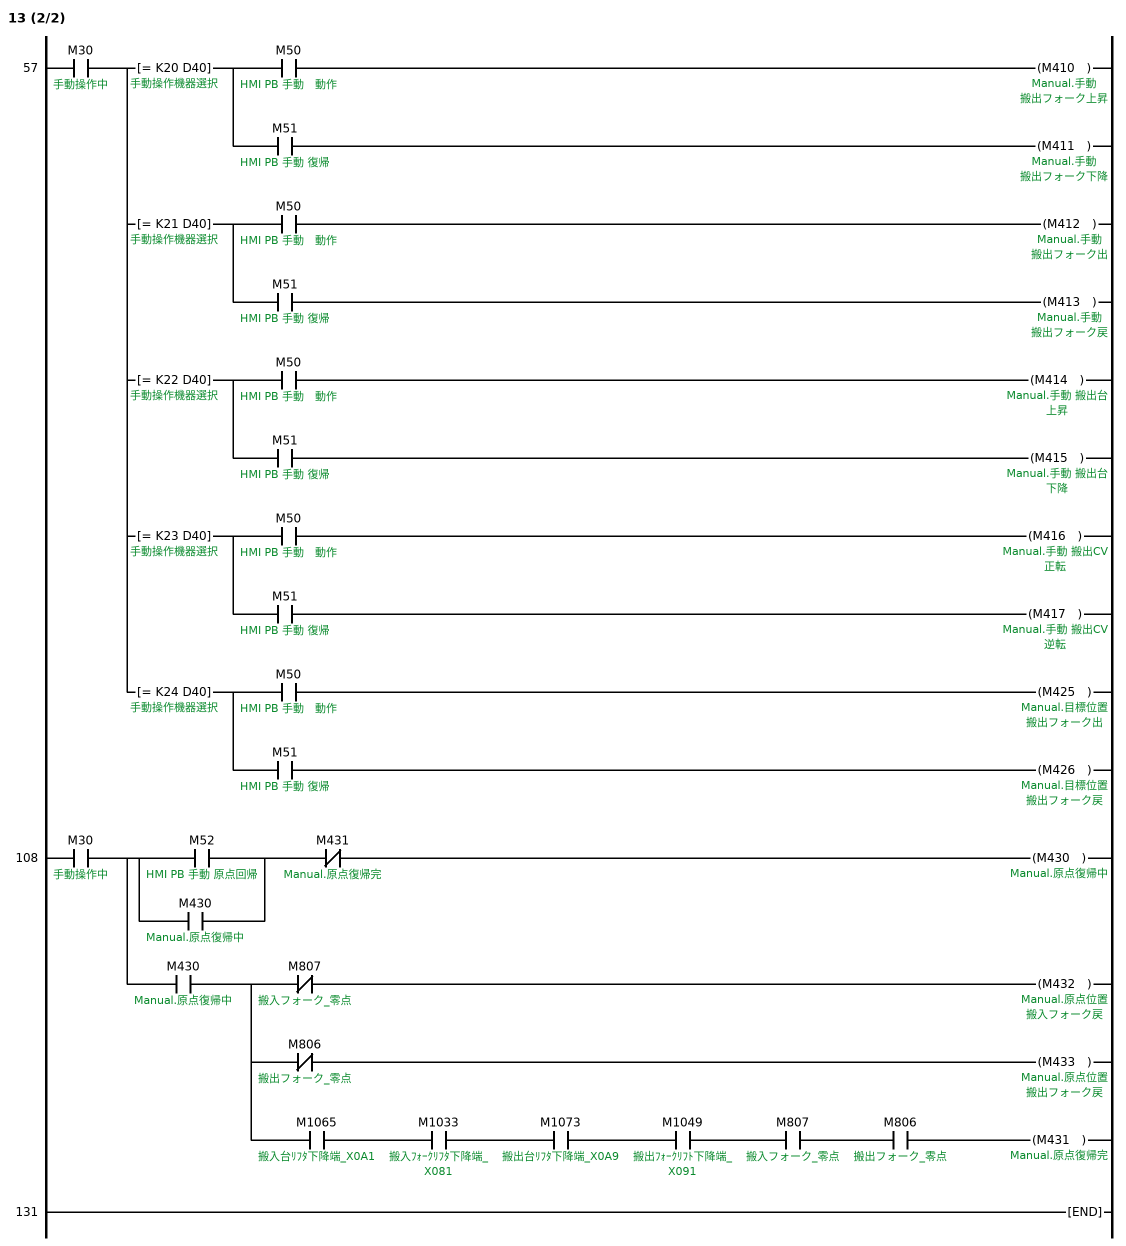
57    LD      M30  ; 手動操作中
      MPS
      AND=    K20 D40  ; 手動操作機器選択
      MPS
      AND     M50  ; HMI PB 手動　動作
      OUT     M410  ; Manual.手動 搬出フォーク上昇
      MPP
      AND     M51  ; HMI PB 手動 復帰
      OUT     M411  ; Manual.手動 搬出フォーク下降
      MRD
      AND=    K21 D40  ; 手動操作機器選択
      MPS
      AND     M50  ; HMI PB 手動　動作
      OUT     M412  ; Manual.手動 搬出フォーク出
      MPP
      AND     M51  ; HMI PB 手動 復帰
      OUT     M413  ; Manual.手動 搬出フォーク戻
      MRD
      AND=    K22 D40  ; 手動操作機器選択
      MPS
      AND     M50  ; HMI PB 手動　動作
      OUT     M414  ; Manual.手動 搬出台 上昇
      MPP
      AND     M51  ; HMI PB 手動 復帰
      OUT     M415  ; Manual.手動 搬出台 下降
      MRD
      AND=    K23 D40  ; 手動操作機器選択
      MPS
      AND     M50  ; HMI PB 手動　動作
      OUT     M416  ; Manual.手動 搬出CV 正転
      MPP
      AND     M51  ; HMI PB 手動 復帰
      OUT     M417  ; Manual.手動 搬出CV 逆転
      MPP
      AND=    K24 D40  ; 手動操作機器選択
      MPS
      AND     M50  ; HMI PB 手動　動作
      OUT     M425  ; Manual.目標位置 搬出フォーク出
      MPP
      AND     M51  ; HMI PB 手動 復帰
      OUT     M426  ; Manual.目標位置 搬出フォーク戻
108   LD      M30  ; 手動操作中
      MPS
      LD      M52  ; HMI PB 手動 原点回帰
      OR      M430  ; Manual.原点復帰中
      ANB
      ANI     M431  ; Manual.原点復帰完
      OUT     M430  ; Manual.原点復帰中
      MPP
      AND     M430  ; Manual.原点復帰中
      MPS
      ANI     M807  ; 搬入フォーク_零点
      OUT     M432  ; Manual.原点位置 搬入フォーク戻
      MRD
      ANI     M806  ; 搬出フォーク_零点
      OUT     M433  ; Manual.原点位置 搬出フォーク戻
      MPP
      AND     M1065  ; 搬入台ﾘﾌﾀ下降端_X0A1
      AND     M1033  ; 搬入ﾌｫｰｸﾘﾌﾀ下降端_X081
      AND     M1073  ; 搬出台ﾘﾌﾀ下降端_X0A9
      AND     M1049  ; 搬出ﾌｫｰｸﾘﾌﾄ下降端_X091
      AND     M807  ; 搬入フォーク_零点
      AND     M806  ; 搬出フォーク_零点
      OUT     M431  ; Manual.原点復帰完
131   END
END_PROGRAM

PROGRAM 20  // INV
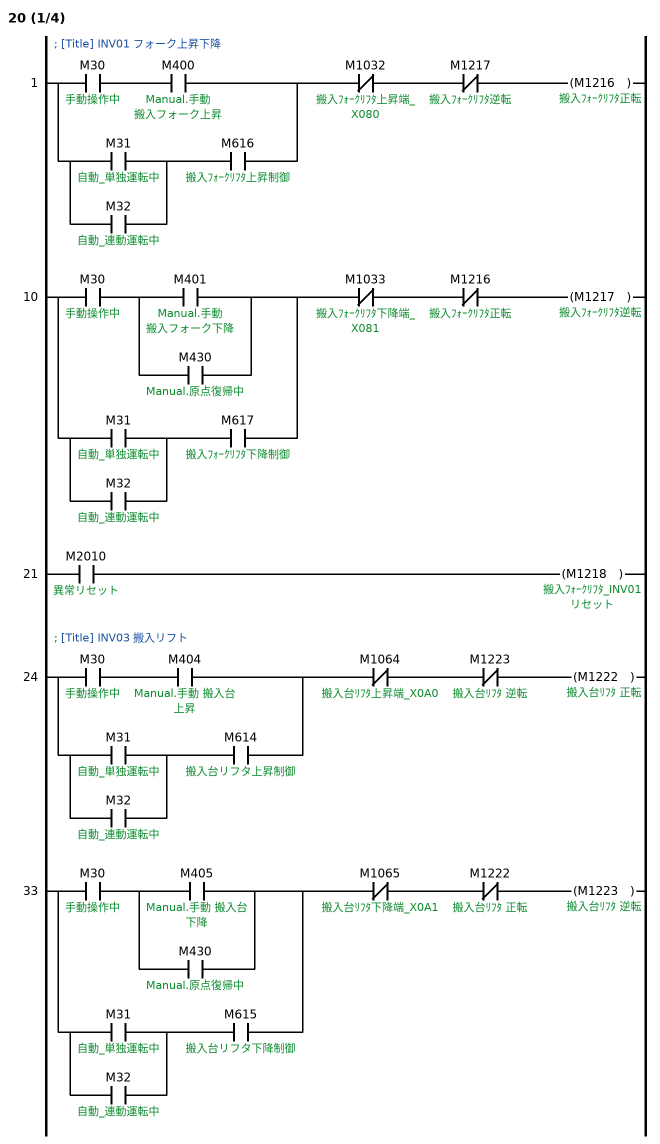
; [Title] INV01 フォーク上昇下降
1     LD      M30  ; 手動操作中
      AND     M400  ; Manual.手動 搬入フォーク上昇
      LD      M31  ; 自動_単独運転中
      OR      M32  ; 自動_連動運転中
      AND     M616  ; 搬入ﾌｫｰｸﾘﾌﾀ上昇制御
      ORB
      ANI     M1032  ; 搬入ﾌｫｰｸﾘﾌﾀ上昇端_X080
      ANI     M1217  ; 搬入ﾌｫｰｸﾘﾌﾀ逆転
      OUT     M1216  ; 搬入ﾌｫｰｸﾘﾌﾀ正転
10    LD      M30  ; 手動操作中
      LD      M401  ; Manual.手動 搬入フォーク下降
      OR      M430  ; Manual.原点復帰中
      ANB
      LD      M31  ; 自動_単独運転中
      OR      M32  ; 自動_連動運転中
      AND     M617  ; 搬入ﾌｫｰｸﾘﾌﾀ下降制御
      ORB
      ANI     M1033  ; 搬入ﾌｫｰｸﾘﾌﾀ下降端_X081
      ANI     M1216  ; 搬入ﾌｫｰｸﾘﾌﾀ正転
      OUT     M1217  ; 搬入ﾌｫｰｸﾘﾌﾀ逆転
21    LD      M2010  ; 異常リセット
      OUT     M1218  ; 搬入ﾌｫｰｸﾘﾌﾀ_INV01 リセット
; [Title] INV03 搬入リフト
24    LD      M30  ; 手動操作中
      AND     M404  ; Manual.手動 搬入台 上昇
      LD      M31  ; 自動_単独運転中
      OR      M32  ; 自動_連動運転中
      AND     M614  ; 搬入台リフタ上昇制御
      ORB
      ANI     M1064  ; 搬入台ﾘﾌﾀ上昇端_X0A0
      ANI     M1223  ; 搬入台ﾘﾌﾀ 逆転
      OUT     M1222  ; 搬入台ﾘﾌﾀ 正転
33    LD      M30  ; 手動操作中
      LD      M405  ; Manual.手動 搬入台 下降
      OR      M430  ; Manual.原点復帰中
      ANB
      LD      M31  ; 自動_単独運転中
      OR      M32  ; 自動_連動運転中
      AND     M615  ; 搬入台リフタ下降制御
      ORB
      ANI     M1065  ; 搬入台ﾘﾌﾀ下降端_X0A1
      ANI     M1222  ; 搬入台ﾘﾌﾀ 正転
      OUT     M1223  ; 搬入台ﾘﾌﾀ 逆転
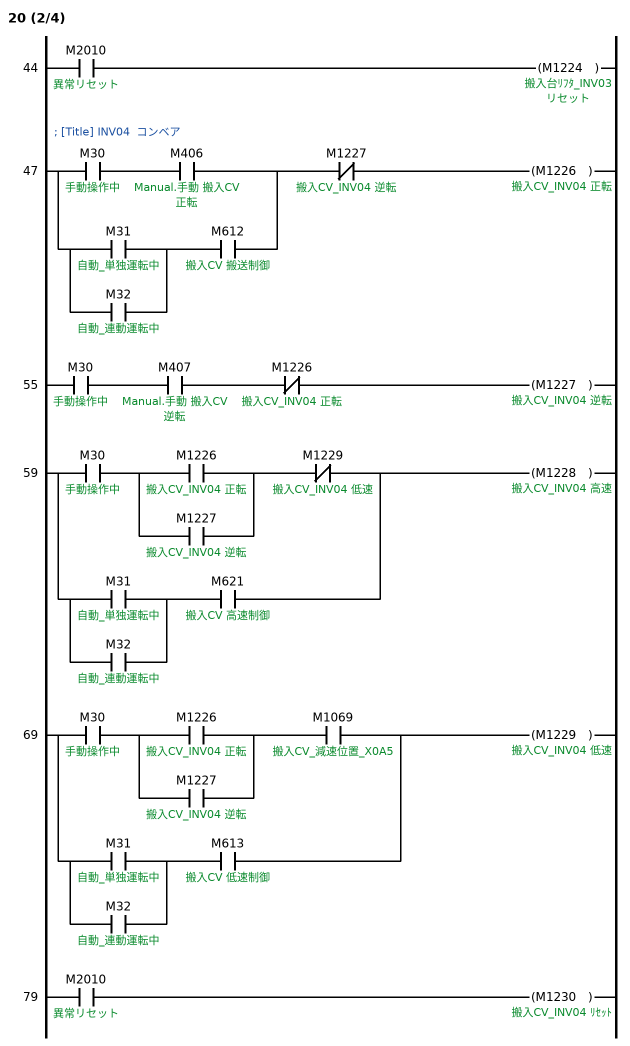
44    LD      M2010  ; 異常リセット
      OUT     M1224  ; 搬入台ﾘﾌﾀ_INV03 リセット
; [Title] INV04  コンベア
47    LD      M30  ; 手動操作中
      AND     M406  ; Manual.手動 搬入CV 正転
      LD      M31  ; 自動_単独運転中
      OR      M32  ; 自動_連動運転中
      AND     M612  ; 搬入CV 搬送制御
      ORB
      ANI     M1227  ; 搬入CV_INV04 逆転
      OUT     M1226  ; 搬入CV_INV04 正転
55    LD      M30  ; 手動操作中
      AND     M407  ; Manual.手動 搬入CV 逆転
      ANI     M1226  ; 搬入CV_INV04 正転
      OUT     M1227  ; 搬入CV_INV04 逆転
59    LD      M30  ; 手動操作中
      LD      M1226  ; 搬入CV_INV04 正転
      OR      M1227  ; 搬入CV_INV04 逆転
      ANB
      ANI     M1229  ; 搬入CV_INV04 低速
      LD      M31  ; 自動_単独運転中
      OR      M32  ; 自動_連動運転中
      AND     M621  ; 搬入CV 高速制御
      ORB
      OUT     M1228  ; 搬入CV_INV04 高速
69    LD      M30  ; 手動操作中
      LD      M1226  ; 搬入CV_INV04 正転
      OR      M1227  ; 搬入CV_INV04 逆転
      ANB
      AND     M1069  ; 搬入CV_減速位置_X0A5
      LD      M31  ; 自動_単独運転中
      OR      M32  ; 自動_連動運転中
      AND     M613  ; 搬入CV 低速制御
      ORB
      OUT     M1229  ; 搬入CV_INV04 低速
79    LD      M2010  ; 異常リセット
      OUT     M1230  ; 搬入CV_INV04 ﾘｾｯﾄ
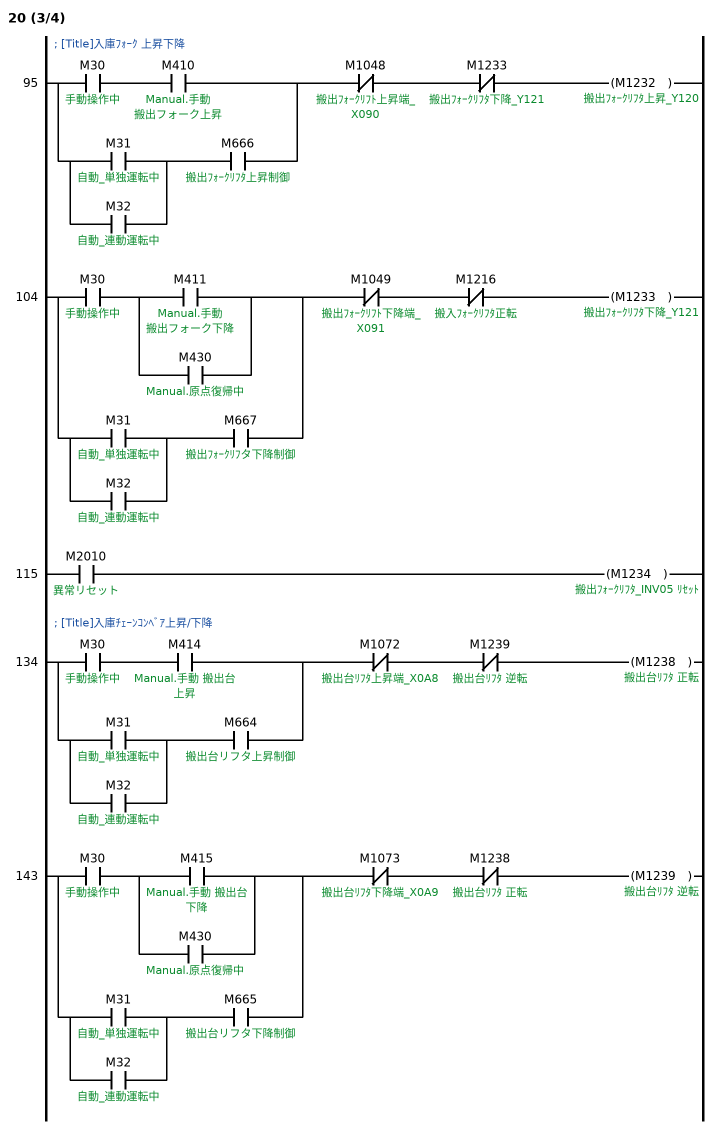
; [Title]入庫ﾌｫｰｸ 上昇下降
95    LD      M30  ; 手動操作中
      AND     M410  ; Manual.手動 搬出フォーク上昇
      LD      M31  ; 自動_単独運転中
      OR      M32  ; 自動_連動運転中
      AND     M666  ; 搬出ﾌｫｰｸﾘﾌﾀ上昇制御
      ORB
      ANI     M1048  ; 搬出ﾌｫｰｸﾘﾌﾄ上昇端_X090
      ANI     M1233  ; 搬出ﾌｫｰｸﾘﾌﾀ下降_Y121
      OUT     M1232  ; 搬出ﾌｫｰｸﾘﾌﾀ上昇_Y120
104   LD      M30  ; 手動操作中
      LD      M411  ; Manual.手動 搬出フォーク下降
      OR      M430  ; Manual.原点復帰中
      ANB
      LD      M31  ; 自動_単独運転中
      OR      M32  ; 自動_連動運転中
      AND     M667  ; 搬出ﾌｫｰｸﾘﾌタ下降制御
      ORB
      ANI     M1049  ; 搬出ﾌｫｰｸﾘﾌﾄ下降端_X091
      ANI     M1216  ; 搬入ﾌｫｰｸﾘﾌﾀ正転
      OUT     M1233  ; 搬出ﾌｫｰｸﾘﾌﾀ下降_Y121
115   LD      M2010  ; 異常リセット
      OUT     M1234  ; 搬出ﾌｫｰｸﾘﾌﾀ_INV05 ﾘｾｯﾄ
; [Title]入庫ﾁｪｰﾝｺﾝﾍﾞｱ上昇/下降
134   LD      M30  ; 手動操作中
      AND     M414  ; Manual.手動 搬出台 上昇
      LD      M31  ; 自動_単独運転中
      OR      M32  ; 自動_連動運転中
      AND     M664  ; 搬出台リフタ上昇制御
      ORB
      ANI     M1072  ; 搬出台ﾘﾌﾀ上昇端_X0A8
      ANI     M1239  ; 搬出台ﾘﾌﾀ 逆転
      OUT     M1238  ; 搬出台ﾘﾌﾀ 正転
143   LD      M30  ; 手動操作中
      LD      M415  ; Manual.手動 搬出台 下降
      OR      M430  ; Manual.原点復帰中
      ANB
      LD      M31  ; 自動_単独運転中
      OR      M32  ; 自動_連動運転中
      AND     M665  ; 搬出台リフタ下降制御
      ORB
      ANI     M1073  ; 搬出台ﾘﾌﾀ下降端_X0A9
      ANI     M1238  ; 搬出台ﾘﾌﾀ 正転
      OUT     M1239  ; 搬出台ﾘﾌﾀ 逆転
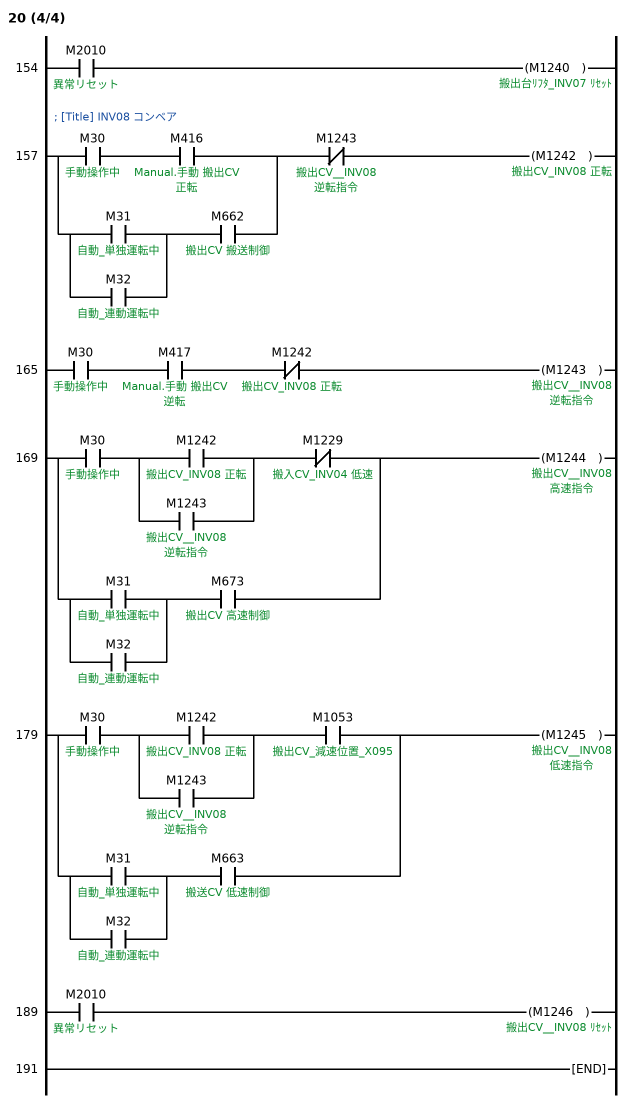
154   LD      M2010  ; 異常リセット
      OUT     M1240  ; 搬出台ﾘﾌﾀ_INV07 ﾘｾｯﾄ
; [Title] INV08 コンベア
157   LD      M30  ; 手動操作中
      AND     M416  ; Manual.手動 搬出CV 正転
      LD      M31  ; 自動_単独運転中
      OR      M32  ; 自動_連動運転中
      AND     M662  ; 搬出CV 搬送制御
      ORB
      ANI     M1243  ; 搬出CV__INV08 逆転指令
      OUT     M1242  ; 搬出CV_INV08 正転
165   LD      M30  ; 手動操作中
      AND     M417  ; Manual.手動 搬出CV 逆転
      ANI     M1242  ; 搬出CV_INV08 正転
      OUT     M1243  ; 搬出CV__INV08 逆転指令
169   LD      M30  ; 手動操作中
      LD      M1242  ; 搬出CV_INV08 正転
      OR      M1243  ; 搬出CV__INV08 逆転指令
      ANB
      ANI     M1229  ; 搬入CV_INV04 低速
      LD      M31  ; 自動_単独運転中
      OR      M32  ; 自動_連動運転中
      AND     M673  ; 搬出CV 高速制御
      ORB
      OUT     M1244  ; 搬出CV__INV08 高速指令
179   LD      M30  ; 手動操作中
      LD      M1242  ; 搬出CV_INV08 正転
      OR      M1243  ; 搬出CV__INV08 逆転指令
      ANB
      AND     M1053  ; 搬出CV_減速位置_X095
      LD      M31  ; 自動_単独運転中
      OR      M32  ; 自動_連動運転中
      AND     M663  ; 搬送CV 低速制御
      ORB
      OUT     M1245  ; 搬出CV__INV08 低速指令
189   LD      M2010  ; 異常リセット
      OUT     M1246  ; 搬出CV__INV08 ﾘｾｯﾄ
191   END
END_PROGRAM

PROGRAM 21  // Fork
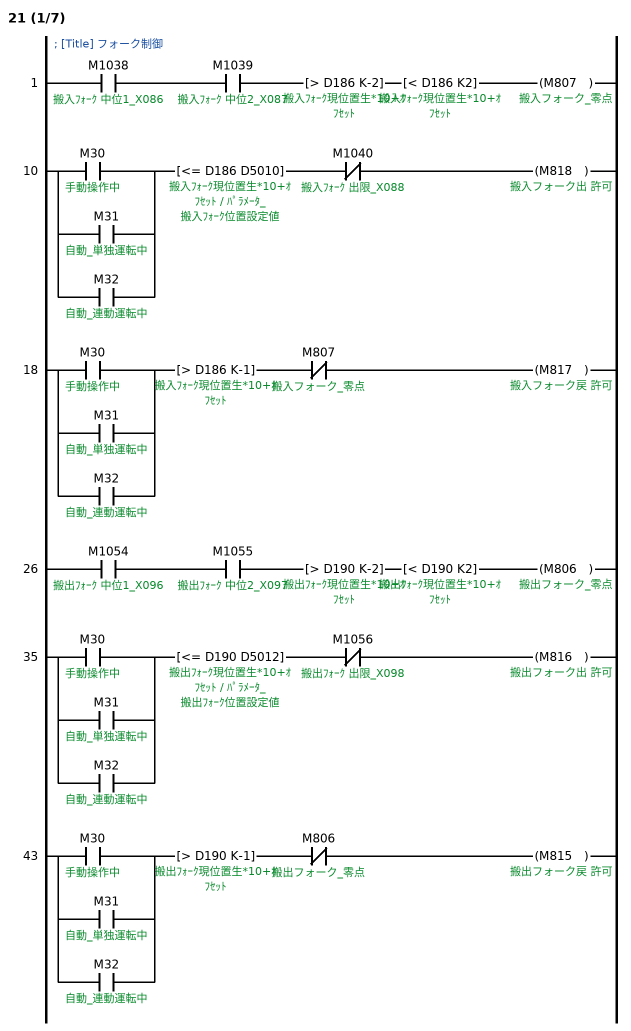
; [Title] フォーク制御
1     LD      M1038  ; 搬入ﾌｫｰｸ 中位1_X086
      AND     M1039  ; 搬入ﾌｫｰｸ 中位2_X087
      AND>    D186 K-2  ; 搬入ﾌｫｰｸ現位置生*10+ｵﾌｾｯﾄ
      AND<    D186 K2  ; 搬入ﾌｫｰｸ現位置生*10+ｵﾌｾｯﾄ
      OUT     M807  ; 搬入フォーク_零点
10    LD      M30  ; 手動操作中
      OR      M31  ; 自動_単独運転中
      OR      M32  ; 自動_連動運転中
      AND<=   D186 D5010  ; 搬入ﾌｫｰｸ現位置生*10+ｵﾌｾｯﾄ / ﾊﾟﾗﾒｰﾀ_搬入ﾌｫｰｸ位置設定値
      ANI     M1040  ; 搬入ﾌｫｰｸ 出限_X088
      OUT     M818  ; 搬入フォーク出 許可
18    LD      M30  ; 手動操作中
      OR      M31  ; 自動_単独運転中
      OR      M32  ; 自動_連動運転中
      AND>    D186 K-1  ; 搬入ﾌｫｰｸ現位置生*10+ｵﾌｾｯﾄ
      ANI     M807  ; 搬入フォーク_零点
      OUT     M817  ; 搬入フォーク戻 許可
26    LD      M1054  ; 搬出ﾌｫｰｸ 中位1_X096
      AND     M1055  ; 搬出ﾌｫｰｸ 中位2_X097
      AND>    D190 K-2  ; 搬出ﾌｫｰｸ現位置生*10+ｵﾌｾｯﾄ
      AND<    D190 K2  ; 搬出ﾌｫｰｸ現位置生*10+ｵﾌｾｯﾄ
      OUT     M806  ; 搬出フォーク_零点
35    LD      M30  ; 手動操作中
      OR      M31  ; 自動_単独運転中
      OR      M32  ; 自動_連動運転中
      AND<=   D190 D5012  ; 搬出ﾌｫｰｸ現位置生*10+ｵﾌｾｯﾄ / ﾊﾟﾗﾒｰﾀ_搬出ﾌｫｰｸ位置設定値
      ANI     M1056  ; 搬出ﾌｫｰｸ 出限_X098
      OUT     M816  ; 搬出フォーク出 許可
43    LD      M30  ; 手動操作中
      OR      M31  ; 自動_単独運転中
      OR      M32  ; 自動_連動運転中
      AND>    D190 K-1  ; 搬出ﾌｫｰｸ現位置生*10+ｵﾌｾｯﾄ
      ANI     M806  ; 搬出フォーク_零点
      OUT     M815  ; 搬出フォーク戻 許可
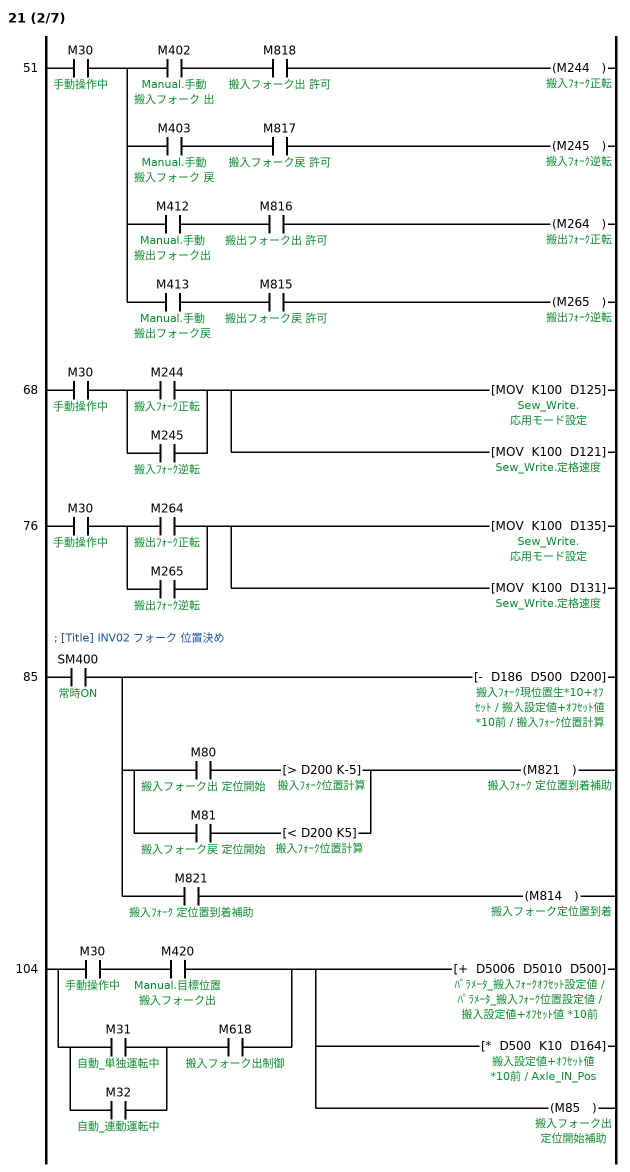
51    LD      M30  ; 手動操作中
      MPS
      AND     M402  ; Manual.手動 搬入フォーク 出
      AND     M818  ; 搬入フォーク出 許可
      OUT     M244  ; 搬入ﾌｫｰｸ正転
      MRD
      AND     M403  ; Manual.手動 搬入フォーク 戻
      AND     M817  ; 搬入フォーク戻 許可
      OUT     M245  ; 搬入ﾌｫｰｸ逆転
      MRD
      AND     M412  ; Manual.手動 搬出フォーク出
      AND     M816  ; 搬出フォーク出 許可
      OUT     M264  ; 搬出ﾌｫｰｸ正転
      MPP
      AND     M413  ; Manual.手動 搬出フォーク戻
      AND     M815  ; 搬出フォーク戻 許可
      OUT     M265  ; 搬出ﾌｫｰｸ逆転
68    LD      M30  ; 手動操作中
      LD      M244  ; 搬入ﾌｫｰｸ正転
      OR      M245  ; 搬入ﾌｫｰｸ逆転
      ANB
      MOV     K100 D125  ; Sew_Write.応用モード設定
      MOV     K100 D121  ; Sew_Write.定格速度
76    LD      M30  ; 手動操作中
      LD      M264  ; 搬出ﾌｫｰｸ正転
      OR      M265  ; 搬出ﾌｫｰｸ逆転
      ANB
      MOV     K100 D135  ; Sew_Write.応用モード設定
      MOV     K100 D131  ; Sew_Write.定格速度
; [Title] INV02 フォーク 位置決め
85    LD      SM400  ; 常時ON
      -       D186 D500 D200  ; 搬入設定値+ｵﾌｾｯﾄ値 *10前 / 搬入ﾌｫｰｸ位置計算
      MPS
      LD      M80  ; 搬入フォーク出 定位開始
      AND>    D200 K-5  ; 搬入ﾌｫｰｸ位置計算
      LD      M81  ; 搬入フォーク戻 定位開始
      AND<    D200 K5  ; 搬入ﾌｫｰｸ位置計算
      ORB
      ANB
      OUT     M821  ; 搬入ﾌｫｰｸ 定位置到着補助
      MPP
      AND     M821  ; 搬入ﾌｫｰｸ 定位置到着補助
      OUT     M814  ; 搬入フォーク定位置到着
104   LD      M30  ; 手動操作中
      AND     M420  ; Manual.目標位置 搬入フォーク出
      LD      M31  ; 自動_単独運転中
      OR      M32  ; 自動_連動運転中
      AND     M618  ; 搬入フォーク出制御
      ORB
      +       D5006 D5010 D500  ; ﾊﾟﾗﾒｰﾀ_搬入ﾌｫｰｸｵﾌｾｯﾄ設定値
      *       D500 K10 D164  ; Axle_IN_Pos
      OUT     M85  ; 搬入フォーク出 定位開始補助
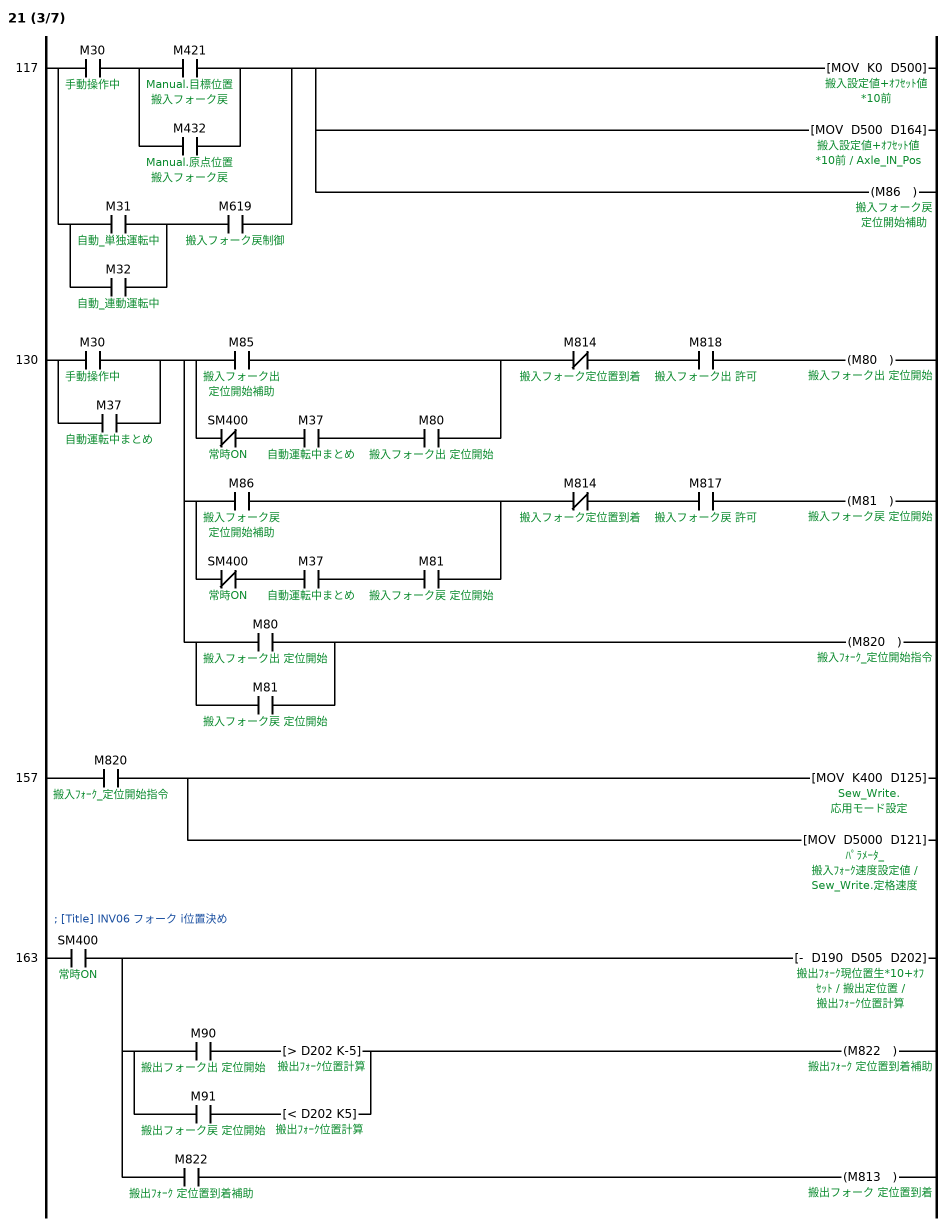
117   LD      M30  ; 手動操作中
      LD      M421  ; Manual.目標位置 搬入フォーク戻
      OR      M432  ; Manual.原点位置 搬入フォーク戻
      ANB
      LD      M31  ; 自動_単独運転中
      OR      M32  ; 自動_連動運転中
      AND     M619  ; 搬入フォーク戻制御
      ORB
      MOV     K0 D500
      MOV     D500 D164
      OUT     M86  ; 搬入フォーク戻 定位開始補助
130   LD      M30  ; 手動操作中
      OR      M37  ; 自動運転中まとめ
      MPS
      LD      M85  ; 搬入フォーク出 定位開始補助
      LDI     SM400  ; 常時ON
      AND     M37  ; 自動運転中まとめ
      AND     M80  ; 搬入フォーク出 定位開始
      ORB
      ANB
      ANI     M814  ; 搬入フォーク定位置到着
      AND     M818  ; 搬入フォーク出 許可
      OUT     M80  ; 搬入フォーク出 定位開始
      MRD
      LD      M86  ; 搬入フォーク戻 定位開始補助
      LDI     SM400  ; 常時ON
      AND     M37  ; 自動運転中まとめ
      AND     M81  ; 搬入フォーク戻 定位開始
      ORB
      ANB
      ANI     M814  ; 搬入フォーク定位置到着
      AND     M817  ; 搬入フォーク戻 許可
      OUT     M81  ; 搬入フォーク戻 定位開始
      MPP
      LD      M80  ; 搬入フォーク出 定位開始
      OR      M81  ; 搬入フォーク戻 定位開始
      ANB
      OUT     M820  ; 搬入ﾌｫｰｸ_定位開始指令
157   LD      M820  ; 搬入ﾌｫｰｸ_定位開始指令
      MOV     K400 D125
      MOV     D5000 D121  ; ﾊﾟﾗﾒｰﾀ_搬入ﾌｫｰｸ速度設定値
; [Title] INV06 フォーク i位置決め
163   LD      SM400  ; 常時ON
      -       D190 D505 D202  ; 搬出定位置 / 搬出ﾌｫｰｸ位置計算
      MPS
      LD      M90  ; 搬出フォーク出 定位開始
      AND>    D202 K-5  ; 搬出ﾌｫｰｸ位置計算
      LD      M91  ; 搬出フォーク戻 定位開始
      AND<    D202 K5  ; 搬出ﾌｫｰｸ位置計算
      ORB
      ANB
      OUT     M822  ; 搬出ﾌｫｰｸ 定位置到着補助
      MPP
      AND     M822  ; 搬出ﾌｫｰｸ 定位置到着補助
      OUT     M813  ; 搬出フォーク 定位置到着
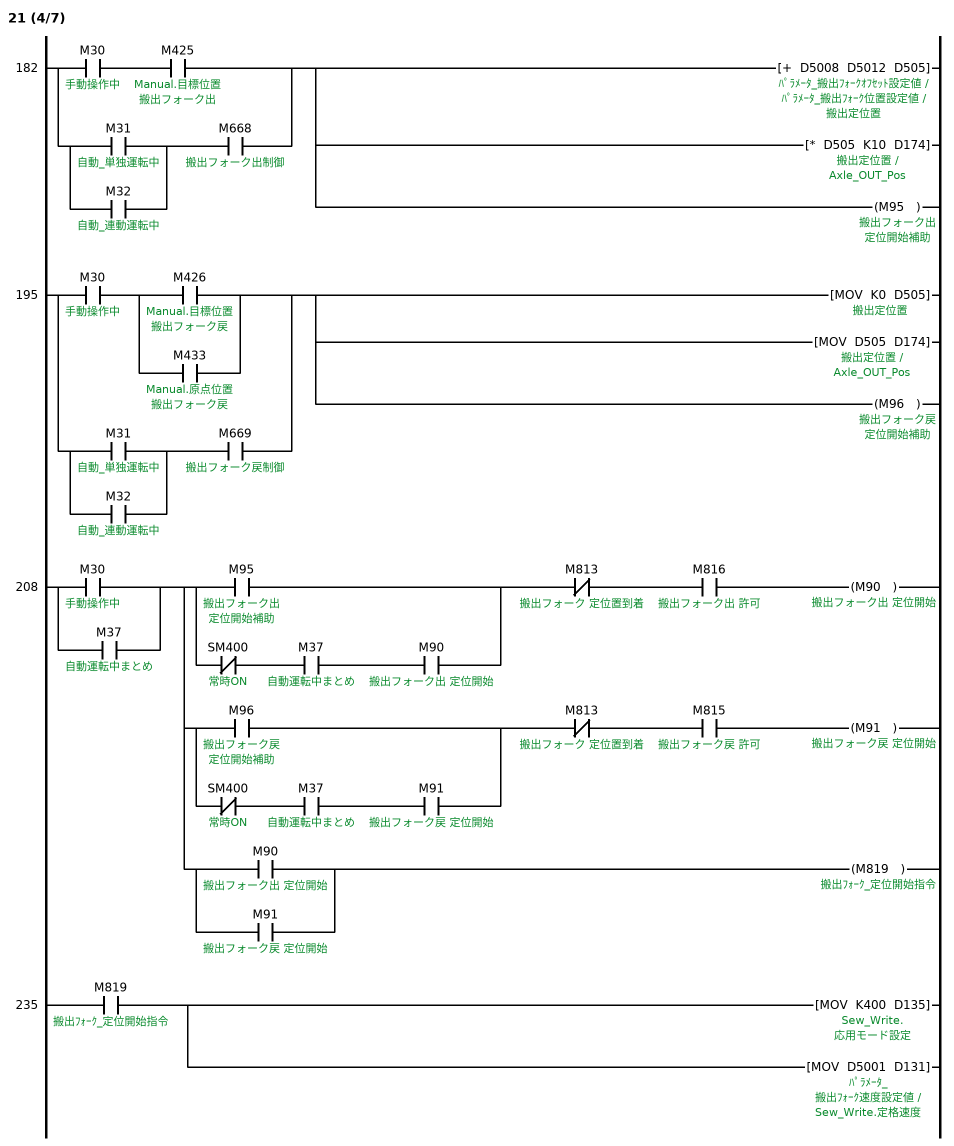
182   LD      M30  ; 手動操作中
      AND     M425  ; Manual.目標位置 搬出フォーク出
      LD      M31  ; 自動_単独運転中
      OR      M32  ; 自動_連動運転中
      AND     M668  ; 搬出フォーク出制御
      ORB
      +       D5008 D5012 D505  ; ﾊﾟﾗﾒｰﾀ_搬出ﾌｫｰｸｵﾌｾｯﾄ設定値
      *       D505 K10 D174  ; Axle_OUT_Pos
      OUT     M95  ; 搬出フォーク出 定位開始補助
195   LD      M30  ; 手動操作中
      LD      M426  ; Manual.目標位置 搬出フォーク戻
      OR      M433  ; Manual.原点位置 搬出フォーク戻
      ANB
      LD      M31  ; 自動_単独運転中
      OR      M32  ; 自動_連動運転中
      AND     M669  ; 搬出フォーク戻制御
      ORB
      MOV     K0 D505
      MOV     D505 D174
      OUT     M96  ; 搬出フォーク戻 定位開始補助
208   LD      M30  ; 手動操作中
      OR      M37  ; 自動運転中まとめ
      MPS
      LD      M95  ; 搬出フォーク出 定位開始補助
      LDI     SM400  ; 常時ON
      AND     M37  ; 自動運転中まとめ
      AND     M90  ; 搬出フォーク出 定位開始
      ORB
      ANB
      ANI     M813  ; 搬出フォーク 定位置到着
      AND     M816  ; 搬出フォーク出 許可
      OUT     M90  ; 搬出フォーク出 定位開始
      MRD
      LD      M96  ; 搬出フォーク戻 定位開始補助
      LDI     SM400  ; 常時ON
      AND     M37  ; 自動運転中まとめ
      AND     M91  ; 搬出フォーク戻 定位開始
      ORB
      ANB
      ANI     M813  ; 搬出フォーク 定位置到着
      AND     M815  ; 搬出フォーク戻 許可
      OUT     M91  ; 搬出フォーク戻 定位開始
      MPP
      LD      M90  ; 搬出フォーク出 定位開始
      OR      M91  ; 搬出フォーク戻 定位開始
      ANB
      OUT     M819  ; 搬出ﾌｫｰｸ_定位開始指令
235   LD      M819  ; 搬出ﾌｫｰｸ_定位開始指令
      MOV     K400 D135
      MOV     D5001 D131  ; ﾊﾟﾗﾒｰﾀ_搬出ﾌｫｰｸ速度設定値
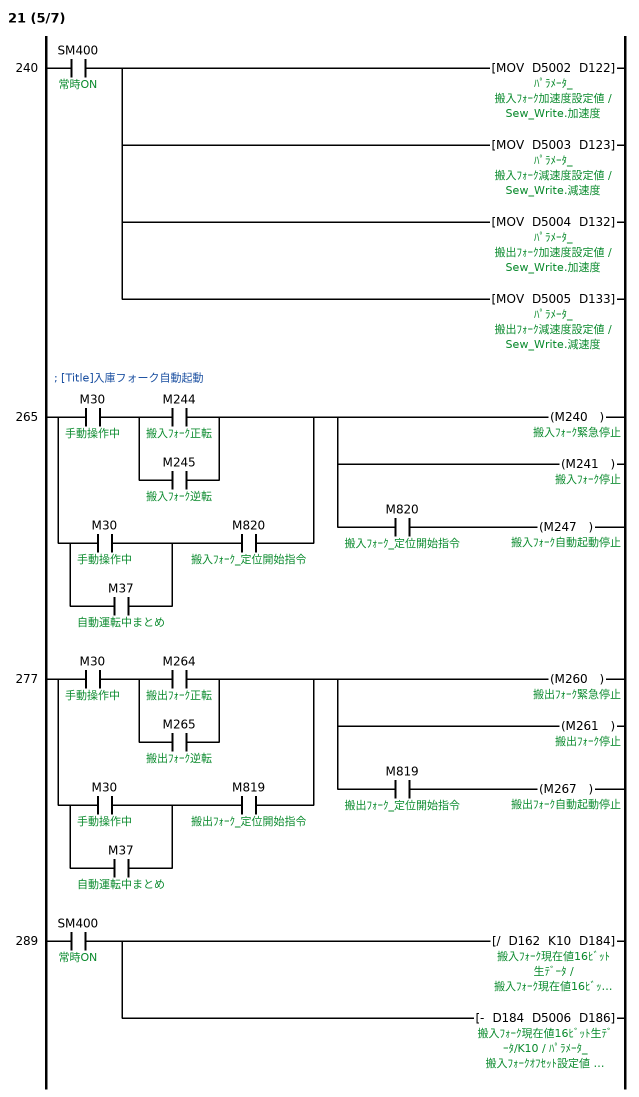
240   LD      SM400  ; 常時ON
      MOV     D5002 D122  ; ﾊﾟﾗﾒｰﾀ_搬入ﾌｫｰｸ加速度設定値 / Sew_Write.加速度
      MOV     D5003 D123  ; ﾊﾟﾗﾒｰﾀ_搬入ﾌｫｰｸ減速度設定値 / Sew_Write.減速度
      MOV     D5004 D132  ; ﾊﾟﾗﾒｰﾀ_搬出ﾌｫｰｸ加速度設定値 / Sew_Write.加速度
      MOV     D5005 D133  ; ﾊﾟﾗﾒｰﾀ_搬出ﾌｫｰｸ減速度設定値 / Sew_Write.減速度
; [Title]入庫フォーク自動起動
265   LD      M30  ; 手動操作中
      LD      M244  ; 搬入ﾌｫｰｸ正転
      OR      M245  ; 搬入ﾌｫｰｸ逆転
      ANB
      LD      M30  ; 手動操作中
      OR      M37  ; 自動運転中まとめ
      AND     M820  ; 搬入ﾌｫｰｸ_定位開始指令
      ORB
      OUT     M240  ; 搬入ﾌｫｰｸ緊急停止
      OUT     M241  ; 搬入ﾌｫｰｸ停止
      AND     M820  ; 搬入ﾌｫｰｸ_定位開始指令
      OUT     M247  ; 搬入ﾌｫｰｸ自動起動停止
277   LD      M30  ; 手動操作中
      LD      M264  ; 搬出ﾌｫｰｸ正転
      OR      M265  ; 搬出ﾌｫｰｸ逆転
      ANB
      LD      M30  ; 手動操作中
      OR      M37  ; 自動運転中まとめ
      AND     M819  ; 搬出ﾌｫｰｸ_定位開始指令
      ORB
      OUT     M260  ; 搬出ﾌｫｰｸ緊急停止
      OUT     M261  ; 搬出ﾌｫｰｸ停止
      AND     M819  ; 搬出ﾌｫｰｸ_定位開始指令
      OUT     M267  ; 搬出ﾌｫｰｸ自動起動停止
289   LD      SM400  ; 常時ON
      /       D162 K10 D184  ; 搬入ﾌｫｰｸ現在値16ﾋﾞｯﾄ生ﾃﾞｰﾀ / 搬入ﾌｫｰｸ現在値16ﾋﾞｯﾄ生ﾃﾞｰﾀ/K10
      -       D184 D5006 D186
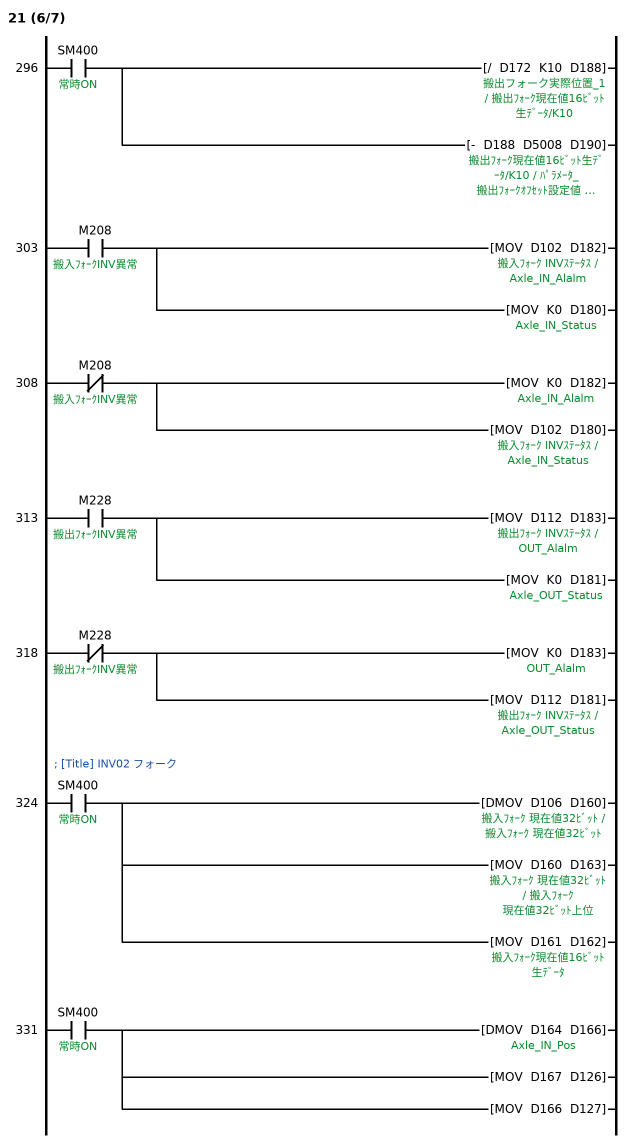
296   LD      SM400  ; 常時ON
      /       D172 K10 D188  ; 搬出フォーク実際位置_1 / 搬出ﾌｫｰｸ現在値16ﾋﾞｯﾄ生ﾃﾞｰﾀ/K10
      -       D188 D5008 D190
303   LD      M208  ; 搬入ﾌｫｰｸINV異常
      MOV     D102 D182  ; 搬入ﾌｫｰｸ INVｽﾃｰﾀｽ / Axle_IN_Alalm
      MOV     K0 D180  ; Axle_IN_Status
308   LDI     M208  ; 搬入ﾌｫｰｸINV異常
      MOV     K0 D182
      MOV     D102 D180
313   LD      M228  ; 搬出ﾌｫｰｸINV異常
      MOV     D112 D183  ; 搬出ﾌｫｰｸ INVｽﾃｰﾀｽ / OUT_Alalm
      MOV     K0 D181  ; Axle_OUT_Status
318   LDI     M228  ; 搬出ﾌｫｰｸINV異常
      MOV     K0 D183
      MOV     D112 D181
; [Title] INV02 フォーク
324   LD      SM400  ; 常時ON
      DMOV    D106 D160  ; 搬入ﾌｫｰｸ 現在値32ﾋﾞｯﾄ / 搬入ﾌｫｰｸ 現在値32ﾋﾞｯﾄ
      MOV     D160 D163  ; 搬入ﾌｫｰｸ 現在値32ﾋﾞｯﾄ上位
      MOV     D161 D162
331   LD      SM400  ; 常時ON
      DMOV    D164 D166
      MOV     D167 D126
      MOV     D166 D127
